  MoveL 7361 to (552.16, 514.95, 128) mm, rotated rx 180 ry 0 rz 160 deg; joints [7.263, 67.715, -20.224, -145.045, 53.083, 157.223]
  Set speed (16.3 mm/s)
  Call Extruder(797.85482)
  MoveL 7362 to (551.52, 517.03, 128) mm, rotated rx -180 ry 0 rz 160 deg; joints [7.506, 67.637, -20.071, -144.797, 53.24, 157.109]
  Call Extruder(805.35406)
  MoveL 7363 to (550.8, 519.07, 128) mm, rotated rx 180 ry 0 rz 160 deg; joints [7.746, 67.545, -19.889, -144.56, 53.407, 157.01]
  Set speed (16.3 mm/s)
  Call Extruder(809.35775)
  MoveL 7364 to (550.38, 520.14, 128) mm, rotated rx 180 ry 0 rz 160 deg; joints [7.874, 67.489, -19.778, -144.438, 53.501, 156.962]
  Set speed (16.2 mm/s)
  Call Extruder(812.97522)
  MoveL 7365 to (549.99, 521.11, 128) mm, rotated rx 180 ry 0 rz 160 deg; joints [7.988, 67.436, -19.673, -144.329, 53.588, 156.922]
  Set speed (16.2 mm/s)
  Call Extruder(817.04856)
  MoveL 7366 to (549.52, 522.18, 128) mm, rotated rx 180 ry 0 rz 160 deg; joints [8.117, 67.37, -19.543, -144.21, 53.691, 156.882]
  Set speed (16.3 mm/s)
  Call Extruder(820.74398)
  MoveL 7367 to (549.08, 523.15, 128) mm, rotated rx 180 ry 0 rz 160 deg; joints [8.233, 67.308, -19.421, -144.103, 53.786, 156.847]
  Set speed (16.3 mm/s)
  Call Extruder(824.78698)
  MoveL 7368 to (548.57, 524.2, 128) mm, rotated rx -180 ry 0 rz 160 deg; joints [8.359, 67.236, -19.278, -143.989, 53.893, 156.814]
  Set speed (16.3 mm/s)
  Call Extruder(830.04096)
  MoveL 7369 to (547.87, 525.55, 128) mm, rotated rx 180 ry 0 rz 160 deg; joints [8.523, 67.135, -19.079, -143.846, 54.037, 156.776]
  Set speed (16.3 mm/s)
  Call Extruder(836.18149)
  MoveL 7370 to (547.01, 527.1, 128) mm, rotated rx 180 ry 0 rz 160 deg; joints [8.712, 67.009, -18.828, -143.684, 54.212, 156.741]
  Set speed (16.3 mm/s)
  Call Extruder(840.06133)
  MoveL 7371 to (546.44, 528.06, 128) mm, rotated rx 180 ry 0 rz 160 deg; joints [8.831, 66.924, -18.66, -143.585, 54.325, 156.723]
  Set speed (16.3 mm/s)
  Call Extruder(844.64327)
  MoveL 7372 to (545.75, 529.18, 128) mm, rotated rx 180 ry 0 rz 160 deg; joints [8.97, 66.819, -18.453, -143.472, 54.463, 156.707]
  Set speed (16.3 mm/s)
  Call Extruder(847.13279)
  MoveL 7373 to (545.36, 529.78, 128) mm, rotated rx -180 ry 0 rz 160 deg; joints [9.045, 66.761, -18.336, -143.412, 54.539, 156.7]
  Set speed (16.3 mm/s)
  Call Extruder(851.62819)
  MoveL 7374 to (544.63, 530.86, 128) mm, rotated rx 180 ry 0 rz 160 deg; joints [9.179, 66.65, -18.117, -143.306, 54.679, 156.692]
  Set speed (16.3 mm/s)
  Call Extruder(855.44742)
  MoveL 7375 to (544, 531.76, 128) mm, rotated rx -180 ry 0 rz 160 deg; joints [9.293, 66.553, -17.924, -143.219, 54.801, 156.688]
  Set speed (16.3 mm/s)
  Call Extruder(859.46697)
  MoveL 7376 to (543.31, 532.69, 128) mm, rotated rx 180 ry 0 rz 160 deg; joints [9.411, 66.446, -17.713, -143.13, 54.931, 156.688]
  Set speed (16.3 mm/s)
  Call Extruder(863.24458)
  MoveL 7377 to (542.65, 533.55, 128) mm, rotated rx 180 ry 0 rz 160 deg; joints [9.522, 66.344, -17.51, -143.049, 55.055, 156.691]
  Set speed (16.3 mm/s)
  Call Extruder(867.09312)
  MoveL 7378 to (541.95, 534.42, 128) mm, rotated rx -180 ry 0 rz 160 deg; joints [9.633, 66.235, -17.295, -142.969, 55.185, 156.698]
  Set speed (16.3 mm/s)
  Call Extruder(870.82681)
  MoveL 7379 to (541.26, 535.24, 128) mm, rotated rx -180 ry 0 rz 160 deg; joints [9.74, 66.128, -17.082, -142.894, 55.311, 156.707]
  Set speed (16.3 mm/s)
  Call Extruder(874.69315)
  MoveL 7380 to (540.53, 536.08, 128) mm, rotated rx 180 ry 0 rz 160 deg; joints [9.85, 66.013, -16.854, -142.818, 55.445, 156.721]
  Set speed (16.3 mm/s)
  Call Extruder(878.56523)
  MoveL 7381 to (539.77, 536.91, 128) mm, rotated rx -180 ry 0 rz 160 deg; joints [9.958, 65.895, -16.619, -142.746, 55.58, 156.737]
  Call Extruder(882.39538)
  MoveL 7382 to (539.02, 537.71, 128) mm, rotated rx -180 ry 0 rz 160 deg; joints [10.065, 65.775, -16.382, -142.676, 55.716, 156.757]
  Call Extruder(886.34677)
  MoveL 7383 to (538.22, 538.52, 128) mm, rotated rx -180 ry 0 rz 160 deg; joints [10.173, 65.649, -16.131, -142.607, 55.858, 156.781]
  Set speed (16.3 mm/s)
  Call Extruder(890.12986)
  MoveL 7384 to (537.43, 539.28, 128) mm, rotated rx 180 ry 0 rz 160 deg; joints [10.276, 65.525, -15.885, -142.543, 55.996, 156.807]
  Call Extruder(893.94691)
  MoveL 7385 to (536.63, 540.03, 128) mm, rotated rx -180 ry 0 rz 160 deg; joints [10.378, 65.398, -15.631, -142.482, 56.136, 156.836]
  Call Extruder(897.84566)
  MoveL 7386 to (535.79, 540.78, 128) mm, rotated rx -180 ry 0 rz 160 deg; joints [10.481, 65.265, -15.367, -142.421, 56.28, 156.869]
  Set speed (16.3 mm/s)
  Call Extruder(901.21524)
  MoveL 7387 to (535.06, 541.42, 128) mm, rotated rx 180 ry 0 rz 160 deg; joints [10.57, 65.148, -15.135, -142.37, 56.407, 156.899]
  Set speed (16.3 mm/s)
  Call Extruder(905.50699)
  MoveL 7388 to (534.11, 542.2, 128) mm, rotated rx -180 ry 0 rz 160 deg; joints [10.68, 64.996, -14.833, -142.309, 56.569, 156.942]
  Set speed (16.3 mm/s)
  Call Extruder(908.78682)
  MoveL 7389 to (533.36, 542.79, 128) mm, rotated rx 180 ry 0 rz 160 deg; joints [10.763, 64.878, -14.597, -142.265, 56.694, 156.978]
  Set speed (16.3 mm/s)
  Call Extruder(913.16892)
  MoveL 7390 to (532.36, 543.56, 128) mm, rotated rx 180 ry 0 rz 160 deg; joints [10.873, 64.718, -14.278, -142.208, 56.862, 157.027]
  Call Extruder(917.07721)
  MoveL 7391 to (531.45, 544.22, 128) mm, rotated rx 180 ry 0 rz 160 deg; joints [10.969, 64.572, -13.988, -142.16, 57.014, 157.075]
  Set speed (16.3 mm/s)
  Call Extruder(920.88896)
  MoveL 7392 to (530.55, 544.85, 128) mm, rotated rx -180 ry 0 rz 160 deg; joints [11.061, 64.428, -13.701, -142.115, 57.163, 157.125]
  Set speed (16.3 mm/s)
  Call Extruder(924.82440)
  MoveL 7393 to (529.6, 545.48, 128) mm, rotated rx 180 ry 0 rz 160 deg; joints [11.155, 64.277, -13.4, -142.072, 57.318, 157.179]
  Set speed (16.3 mm/s)
  Call Extruder(928.58871)
  MoveL 7394 to (528.69, 546.06, 128) mm, rotated rx -180 ry 0 rz 160 deg; joints [11.243, 64.13, -13.108, -142.033, 57.467, 157.233]
  Set speed (16.3 mm/s)
  Call Extruder(932.50029)
  MoveL 7395 to (527.73, 546.64, 128) mm, rotated rx -180 ry 0 rz 160 deg; joints [11.333, 63.976, -12.8, -141.994, 57.622, 157.293]
  Set speed (16.3 mm/s)
  Call Extruder(936.32920)
  MoveL 7396 to (526.77, 547.2, 128) mm, rotated rx 180 ry 0 rz 160 deg; joints [11.419, 63.823, -12.495, -141.96, 57.775, 157.353]
  Set speed (16.3 mm/s)
  Call Extruder(939.88963)
  MoveL 7397 to (525.88, 547.7, 128) mm, rotated rx -180 ry 0 rz 160 deg; joints [11.498, 63.679, -12.208, -141.929, 57.918, 157.412]
  Set speed (16.3 mm/s)
  Call Extruder(946.13638)
  MoveL 7398 to (524.28, 548.53, 128) mm, rotated rx 180 ry 0 rz 160 deg; joints [11.632, 63.424, -11.698, -141.881, 58.17, 157.52]
  Call Extruder(951.88293)
  MoveL 7399 to (522.79, 549.25, 128) mm, rotated rx 180 ry 0 rz 160 deg; joints [11.751, 63.185, -11.22, -141.843, 58.404, 157.625]
  Set speed (16.3 mm/s)
  Call Extruder(959.39188)
  MoveL 7400 to (520.81, 550.12, 128) mm, rotated rx 180 ry 0 rz 160 deg; joints [11.901, 62.867, -10.585, -141.8, 58.71, 157.77]
  Call Extruder(967.32682)
  MoveL 7401 to (518.68, 550.95, 128) mm, rotated rx 180 ry 0 rz 160 deg; joints [12.051, 62.526, -9.902, -141.766, 59.035, 157.933]
  Set speed (16.3 mm/s)
  Call Extruder(974.78424)
  MoveL 7402 to (516.64, 551.64, 128) mm, rotated rx 180 ry 0 rz 160 deg; joints [12.184, 62.2, -9.25, -141.743, 59.341, 158.095]
  Set speed (16.2 mm/s)
  Call Extruder(978.78034)
  MoveL 7403 to (515.54, 551.98, 128) mm, rotated rx -180 ry 0 rz 160 deg; joints [12.252, 62.024, -8.897, -141.734, 59.505, 158.185]
  Set speed (16.3 mm/s)
  Call Extruder(982.65084)
  MoveL 7404 to (514.48, 552.3, 128) mm, rotated rx 180 ry 0 rz 160 deg; joints [12.316, 61.854, -8.554, -141.727, 59.664, 158.273]
  Call Extruder(985.91733)
  MoveL 7405 to (513.56, 552.54, 128) mm, rotated rx -180 ry 0 rz 160 deg; joints [12.368, 61.708, -8.262, -141.725, 59.798, 158.351]
  Set speed (16.2 mm/s)
  Call Extruder(990.16839)
  MoveL 7406 to (512.38, 552.83, 128) mm, rotated rx -180 ry 0 rz 160 deg; joints [12.434, 61.518, -7.881, -141.723, 59.973, 158.452]
  Set speed (16.3 mm/s)
  Call Extruder(998.02753)
  MoveL 7407 to (510.16, 553.3, 128) mm, rotated rx 180 ry 0 rz 160 deg; joints [12.548, 61.165, -7.171, -141.727, 60.295, 158.646]
  Set speed (16.3 mm/s)
  Call Extruder(1005.81110)
  MoveL 7408 to (507.95, 553.68, 128) mm, rotated rx 180 ry 0 rz 160 deg; joints [12.652, 60.812, -6.461, -141.742, 60.612, 158.845]
  Call Extruder(1013.42033)
  MoveL 7409 to (505.77, 553.95, 128) mm, rotated rx -180 ry 0 rz 160 deg; joints [12.743, 60.464, -5.762, -141.766, 60.921, 159.047]
  Set speed (16.3 mm/s)
  Call Extruder(1021.17666)
  MoveL 7410 to (503.55, 554.15, 128) mm, rotated rx 180 ry 0 rz 160 deg; joints [12.827, 60.109, -5.047, -141.799, 61.234, 159.258]
  Set speed (16.3 mm/s)
  Call Extruder(1028.91579)
  MoveL 7411 to (501.32, 554.25, 128) mm, rotated rx 180 ry 0 rz 160 deg; joints [12.9, 59.754, -4.33, -141.843, 61.544, 159.475]
  Set speed (16.3 mm/s)
  Call Extruder(1036.52400)
  MoveL 7412 to (499.12, 554.25, 128) mm, rotated rx 180 ry 0 rz 160 deg; joints [12.962, 59.405, -3.625, -141.895, 61.846, 159.694]
  Set speed (10.0 mm/s)
  MoveL 7413 to (499.12, 554.25, 132) mm, rotated rx 180 ry 0 rz 160 deg; joints [12.962, 58.806, -3.422, -141.763, 61.534, 159.416]
  Set speed (120.0 mm/s)
  MoveL 7414 to (499.15, 552.4, 132) mm, rotated rx 180 ry 0 rz 160 deg; joints [12.736, 58.744, -3.297, -142.025, 61.505, 159.575]
  Set speed (16.4 mm/s)
  Call Extruder(1043.97760)
  MoveL 7415 to (496.99, 552.32, 132) mm, rotated rx 180 ry 0 rz 160 deg; joints [12.786, 58.398, -2.602, -142.088, 61.797, 159.793]
  Set speed (16.4 mm/s)
  Call Extruder(1051.39615)
  MoveL 7416 to (494.85, 552.15, 132) mm, rotated rx 180 ry 0 rz 160 deg; joints [12.825, 58.055, -1.913, -142.16, 62.084, 160.015]
  Call Extruder(1058.70817)
  MoveL 7417 to (492.74, 551.9, 132) mm, rotated rx 180 ry 0 rz 160 deg; joints [12.853, 57.719, -1.235, -142.24, 62.364, 160.237]
  Set speed (16.4 mm/s)
  Call Extruder(1066.06150)
  MoveL 7418 to (490.64, 551.56, 132) mm, rotated rx -180 ry 0 rz 160 deg; joints [12.871, 57.381, -0.555, -142.331, 62.64, 160.465]
  Set speed (16.4 mm/s)
  Call Extruder(1073.73360)
  MoveL 7419 to (488.45, 551.12, 132) mm, rotated rx 180 ry 0 rz 160 deg; joints [12.878, 57.032, 0.149, -142.435, 62.924, 160.705]
  Set speed (16.4 mm/s)
  Call Extruder(1077.22198)
  MoveL 7420 to (487.47, 550.88, 132) mm, rotated rx -180 ry 0 rz 160 deg; joints [12.876, 56.874, 0.467, -142.486, 63.051, 160.816]
  Call Extruder(1080.67093)
  MoveL 7421 to (486.5, 550.64, 132) mm, rotated rx -180 ry 0 rz 160 deg; joints [12.873, 56.719, 0.781, -142.538, 63.175, 160.925]
  Set speed (16.4 mm/s)
  Call Extruder(1084.57071)
  MoveL 7422 to (485.41, 550.33, 132) mm, rotated rx -180 ry 0 rz 160 deg; joints [12.866, 56.545, 1.134, -142.6, 63.314, 161.05]
  Call Extruder(1088.21611)
  MoveL 7423 to (484.4, 550.03, 132) mm, rotated rx 180 ry 0 rz 160 deg; joints [12.857, 56.382, 1.462, -142.66, 63.443, 161.167]
  Set speed (16.4 mm/s)
  Call Extruder(1095.48451)
  MoveL 7424 to (482.4, 549.36, 132) mm, rotated rx 180 ry 0 rz 160 deg; joints [12.831, 56.061, 2.112, -142.787, 63.697, 161.402]
  Set speed (16.4 mm/s)
  Call Extruder(1099.40980)
  MoveL 7425 to (481.33, 548.96, 132) mm, rotated rx 180 ry 0 rz 160 deg; joints [12.811, 55.889, 2.46, -142.86, 63.83, 161.529]
  Set speed (16.4 mm/s)
  Call Extruder(1103.58260)
  MoveL 7426 to (480.21, 548.52, 132) mm, rotated rx 180 ry 0 rz 160 deg; joints [12.788, 55.708, 2.827, -142.94, 63.971, 161.665]
  Set speed (16.3 mm/s)
  Call Extruder(1108.58819)
  MoveL 7427 to (478.87, 547.96, 132) mm, rotated rx -180 ry 0 rz 160 deg; joints [12.755, 55.493, 3.263, -143.04, 64.137, 161.828]
  Set speed (16.4 mm/s)
  Call Extruder(1114.05266)
  MoveL 7428 to (477.43, 547.3, 132) mm, rotated rx 180 ry 0 rz 160 deg; joints [12.712, 55.26, 3.734, -143.154, 64.315, 162.007]
  Set speed (16.4 mm/s)
  Call Extruder(1117.85423)
  MoveL 7429 to (476.44, 546.81, 132) mm, rotated rx -180 ry 0 rz 160 deg; joints [12.678, 55.1, 4.06, -143.237, 64.437, 162.132]
  Set speed (16.4 mm/s)
  Call Extruder(1121.57728)
  MoveL 7430 to (475.48, 546.32, 132) mm, rotated rx 180 ry 0 rz 160 deg; joints [12.642, 54.945, 4.375, -143.321, 64.554, 162.255]
  Set speed (16.4 mm/s)
  Call Extruder(1124.36398)
  MoveL 7431 to (474.77, 545.93, 132) mm, rotated rx -180 ry 0 rz 160 deg; joints [12.613, 54.829, 4.61, -143.385, 64.641, 162.346]
  Set speed (16.4 mm/s)
  Call Extruder(1128.80316)
  MoveL 7432 to (473.65, 545.3, 132) mm, rotated rx 180 ry 0 rz 160 deg; joints [12.564, 54.647, 4.98, -143.49, 64.777, 162.493]
  Call Extruder(1132.57278)
  MoveL 7433 to (472.71, 544.74, 132) mm, rotated rx -180 ry 0 rz 160 deg; joints [12.518, 54.494, 5.291, -143.582, 64.891, 162.617]
  Set speed (16.4 mm/s)
  Call Extruder(1136.28054)
  MoveL 7434 to (471.79, 544.17, 132) mm, rotated rx -180 ry 0 rz 160 deg; joints [12.471, 54.346, 5.593, -143.675, 65.001, 162.739]
  Call Extruder(1139.90076)
  MoveL 7435 to (470.92, 543.59, 132) mm, rotated rx 180 ry 0 rz 160 deg; joints [12.421, 54.202, 5.885, -143.768, 65.106, 162.858]
  Set speed (16.4 mm/s)
  Call Extruder(1143.59875)
  MoveL 7436 to (470.03, 542.99, 132) mm, rotated rx 180 ry 0 rz 160 deg; joints [12.368, 54.057, 6.181, -143.865, 65.211, 162.979]
  Set speed (16.4 mm/s)
  Call Extruder(1147.38632)
  MoveL 7437 to (469.13, 542.35, 132) mm, rotated rx -180 ry 0 rz 160 deg; joints [12.31, 53.911, 6.479, -143.968, 65.317, 163.103]
  Set speed (16.4 mm/s)
  Call Extruder(1150.96414)
  MoveL 7438 to (468.3, 541.73, 132) mm, rotated rx 180 ry 0 rz 160 deg; joints [12.253, 53.774, 6.758, -144.066, 65.416, 163.22]
  Set speed (16.4 mm/s)
  Call Extruder(1154.80847)
  MoveL 7439 to (467.42, 541.05, 132) mm, rotated rx 180 ry 0 rz 160 deg; joints [12.188, 53.629, 7.054, -144.174, 65.519, 163.346]
  Call Extruder(1158.41047)
  MoveL 7440 to (466.61, 540.39, 132) mm, rotated rx 180 ry 0 rz 160 deg; joints [12.124, 53.495, 7.327, -144.279, 65.614, 163.463]
  Call Extruder(1162.10973)
  MoveL 7441 to (465.79, 539.69, 132) mm, rotated rx -180 ry 0 rz 160 deg; joints [12.056, 53.36, 7.604, -144.387, 65.71, 163.583]
  Set speed (16.4 mm/s)
  Call Extruder(1165.90163)
  MoveL 7442 to (464.96, 538.97, 132) mm, rotated rx 180 ry 0 rz 160 deg; joints [11.984, 53.222, 7.884, -144.501, 65.806, 163.705]
  Set speed (16.4 mm/s)
  Call Extruder(1169.28030)
  MoveL 7443 to (464.24, 538.31, 132) mm, rotated rx 180 ry 0 rz 160 deg; joints [11.916, 53.102, 8.13, -144.605, 65.889, 163.814]
  Set speed (16.4 mm/s)
  Call Extruder(1172.26831)
  MoveL 7444 to (463.61, 537.71, 132) mm, rotated rx -180 ry 0 rz 160 deg; joints [11.854, 52.998, 8.344, -144.698, 65.961, 163.91]
  Set speed (16.4 mm/s)
  Call Extruder(1176.91926)
  MoveL 7445 to (462.65, 536.76, 132) mm, rotated rx -180 ry 0 rz 160 deg; joints [11.754, 52.838, 8.671, -144.846, 66.07, 164.059]
  Set speed (16.4 mm/s)
  Call Extruder(1180.58115)
  MoveL 7446 to (461.91, 535.99, 132) mm, rotated rx 180 ry 0 rz 160 deg; joints [11.673, 52.714, 8.925, -144.965, 66.154, 164.175]
  Set speed (16.4 mm/s)
  Call Extruder(1184.31373)
  MoveL 7447 to (461.17, 535.2, 132) mm, rotated rx 180 ry 0 rz 160 deg; joints [11.587, 52.59, 9.178, -145.088, 66.237, 164.293]
  Set speed (16.4 mm/s)
  Call Extruder(1187.19569)
  MoveL 7448 to (460.62, 534.57, 132) mm, rotated rx -180 ry 0 rz 160 deg; joints [11.518, 52.496, 9.371, -145.185, 66.299, 164.383]
  Set speed (16.4 mm/s)
  Call Extruder(1191.17044)
  MoveL 7449 to (459.87, 533.7, 132) mm, rotated rx 180 ry 0 rz 160 deg; joints [11.421, 52.369, 9.632, -145.321, 66.383, 164.507]
  Set speed (16.4 mm/s)
  Call Extruder(1195.44747)
  MoveL 7450 to (459.08, 532.74, 132) mm, rotated rx -180 ry 0 rz 160 deg; joints [11.313, 52.235, 9.906, -145.469, 66.47, 164.64]
  Set speed (16.4 mm/s)
  Call Extruder(1199.06168)
  MoveL 7451 to (458.43, 531.91, 132) mm, rotated rx 180 ry 0 rz 160 deg; joints [11.219, 52.124, 10.133, -145.597, 66.541, 164.751]
  Call Extruder(1202.74625)
  MoveL 7452 to (457.79, 531.06, 132) mm, rotated rx 180 ry 0 rz 160 deg; joints [11.121, 52.014, 10.359, -145.729, 66.611, 164.864]
  Set speed (16.4 mm/s)
  Call Extruder(1206.43074)
  MoveL 7453 to (457.17, 530.19, 132) mm, rotated rx 180 ry 0 rz 160 deg; joints [11.02, 51.906, 10.581, -145.863, 66.679, 164.975]
  Set speed (16.4 mm/s)
  Call Extruder(1210.21210)
  MoveL 7454 to (456.55, 529.29, 132) mm, rotated rx -180 ry 0 rz 160 deg; joints [10.913, 51.798, 10.803, -146.002, 66.746, 165.089]
  Set speed (16.4 mm/s)
  Call Extruder(1213.92244)
  MoveL 7455 to (455.95, 528.39, 132) mm, rotated rx 180 ry 0 rz 160 deg; joints [10.806, 51.695, 11.015, -146.141, 66.809, 165.2]
  Set speed (16.4 mm/s)
  Call Extruder(1217.52902)
  MoveL 7456 to (455.39, 527.51, 132) mm, rotated rx -180 ry 0 rz 160 deg; joints [10.7, 51.597, 11.217, -146.277, 66.868, 165.306]
  Set speed (16.4 mm/s)
  Call Extruder(1221.90125)
  MoveL 7457 to (454.74, 526.42, 132) mm, rotated rx -180 ry 0 rz 160 deg; joints [10.568, 51.482, 11.454, -146.445, 66.936, 165.434]
  Call Extruder(1228.58017)
  MoveL 7458 to (453.79, 524.73, 132) mm, rotated rx -180 ry 0 rz 160 deg; joints [10.359, 51.313, 11.802, -146.706, 67.033, 165.627]
  Set speed (16.4 mm/s)
  Call Extruder(1232.29007)
  MoveL 7459 to (453.3, 523.77, 132) mm, rotated rx -180 ry 0 rz 160 deg; joints [10.241, 51.223, 11.987, -146.853, 67.083, 165.732]
  Call Extruder(1236.08269)
  MoveL 7460 to (452.81, 522.79, 132) mm, rotated rx -180 ry 0 rz 160 deg; joints [10.117, 51.134, 12.17, -147.005, 67.132, 165.839]
  Set speed (16.4 mm/s)
  Call Extruder(1243.24840)
  MoveL 7461 to (451.94, 520.9, 132) mm, rotated rx 180 ry 0 rz 160 deg; joints [9.876, 50.974, 12.5, -147.297, 67.216, 166.037]
  Set speed (16.4 mm/s)
  Call Extruder(1247.17185)
  MoveL 7462 to (451.5, 519.85, 132) mm, rotated rx -180 ry 0 rz 160 deg; joints [9.741, 50.891, 12.67, -147.459, 67.258, 166.143]
  Set speed (16.4 mm/s)
  Call Extruder(1250.87077)
  MoveL 7463 to (451.1, 518.85, 132) mm, rotated rx 180 ry 0 rz 160 deg; joints [9.612, 50.815, 12.827, -147.613, 67.295, 166.243]
  Set speed (16.4 mm/s)
  Call Extruder(1254.56538)
  MoveL 7464 to (450.73, 517.85, 132) mm, rotated rx 180 ry 0 rz 160 deg; joints [9.481, 50.744, 12.974, -147.768, 67.328, 166.34]
  Set speed (16.4 mm/s)
  Call Extruder(1258.09802)
  MoveL 7465 to (450.39, 516.88, 132) mm, rotated rx 180 ry 0 rz 160 deg; joints [9.354, 50.677, 13.112, -147.917, 67.358, 166.432]
  Set speed (16.4 mm/s)
  Call Extruder(1261.95788)
  MoveL 7466 to (450.05, 515.82, 132) mm, rotated rx 180 ry 0 rz 160 deg; joints [9.214, 50.608, 13.254, -148.082, 67.387, 166.531]
  Set speed (16.4 mm/s)
  Call Extruder(1265.49475)
  MoveL 7467 to (449.74, 514.84, 132) mm, rotated rx -180 ry 0 rz 160 deg; joints [9.084, 50.547, 13.38, -148.233, 67.413, 166.621]
  Set speed (16.4 mm/s)
  Call Extruder(1272.94487)
  MoveL 7468 to (449.17, 512.75, 132) mm, rotated rx -180 ry 0 rz 160 deg; joints [8.804, 50.429, 13.625, -148.555, 67.456, 166.806]
  Set speed (16.4 mm/s)
  Call Extruder(1280.31638)
  MoveL 7469 to (448.69, 510.67, 132) mm, rotated rx -180 ry 0 rz 160 deg; joints [8.521, 50.324, 13.842, -148.878, 67.488, 166.984]
  Set speed (16.4 mm/s)
  Call Extruder(1287.84373)
  MoveL 7470 to (448.29, 508.52, 132) mm, rotated rx 180 ry 0 rz 160 deg; joints [8.226, 50.229, 14.038, -149.21, 67.508, 167.159]
  Call Extruder(1295.22150)
  MoveL 7471 to (447.99, 506.4, 132) mm, rotated rx 180 ry 0 rz 160 deg; joints [7.933, 50.15, 14.202, -149.538, 67.517, 167.324]
  Set speed (16.4 mm/s)
  Call Extruder(1302.60966)
  MoveL 7472 to (447.77, 504.27, 132) mm, rotated rx -180 ry 0 rz 160 deg; joints [7.635, 50.082, 14.341, -149.867, 67.514, 167.484]
  Set speed (16.4 mm/s)
  Call Extruder(1309.81071)
  MoveL 7473 to (447.64, 502.18, 132) mm, rotated rx 180 ry 0 rz 160 deg; joints [7.342, 50.03, 14.45, -150.189, 67.499, 167.633]
  Set speed (16.4 mm/s)
  Call Extruder(1317.28696)
  MoveL 7474 to (447.59, 500.01, 132) mm, rotated rx -180 ry 0 rz 160 deg; joints [7.034, 49.988, 14.537, -150.524, 67.473, 167.781]
  Set speed (16.4 mm/s)
  Call Extruder(1324.02628)
  MoveL 7475 to (447.63, 498.06, 132) mm, rotated rx 180 ry 0 rz 160 deg; joints [6.755, 49.962, 14.591, -150.824, 67.439, 167.909]
  Set speed (16.4 mm/s)
  Call Extruder(1330.58179)
  MoveL 7476 to (447.74, 496.16, 132) mm, rotated rx 180 ry 0 rz 160 deg; joints [6.483, 49.947, 14.622, -151.116, 67.396, 168.028]
  Set speed (16.4 mm/s)
  Call Extruder(1337.23196)
  MoveL 7477 to (447.91, 494.24, 132) mm, rotated rx -180 ry 0 rz 160 deg; joints [6.206, 49.941, 14.634, -151.41, 67.344, 168.144]
  Call Extruder(1343.87995)
  MoveL 7478 to (448.16, 492.32, 132) mm, rotated rx 180 ry 0 rz 160 deg; joints [5.93, 49.947, 14.621, -151.703, 67.282, 168.254]
  Set speed (16.4 mm/s)
  Call Extruder(1350.61226)
  MoveL 7479 to (448.48, 490.4, 132) mm, rotated rx 180 ry 0 rz 160 deg; joints [5.65, 49.964, 14.586, -151.996, 67.209, 168.36]
  Set speed (16.4 mm/s)
  Call Extruder(1357.16591)
  MoveL 7480 to (448.86, 488.53, 132) mm, rotated rx -180 ry 0 rz 160 deg; joints [5.379, 49.991, 14.531, -152.278, 67.13, 168.457]
  Set speed (16.4 mm/s)
  Call Extruder(1363.73554)
  MoveL 7481 to (449.31, 486.68, 132) mm, rotated rx 180 ry 0 rz 160 deg; joints [5.109, 50.028, 14.455, -152.558, 67.041, 168.549]
  Set speed (16.4 mm/s)
  Call Extruder(1370.46103)
  MoveL 7482 to (449.85, 484.8, 132) mm, rotated rx -180 ry 0 rz 160 deg; joints [4.835, 50.076, 14.354, -152.84, 66.94, 168.637]
  Call Extruder(1377.10545)
  MoveL 7483 to (450.44, 482.97, 132) mm, rotated rx 180 ry 0 rz 160 deg; joints [4.567, 50.135, 14.233, -153.114, 66.832, 168.719]
  Set speed (16.4 mm/s)
  Call Extruder(1383.92639)
  MoveL 7484 to (451.12, 481.11, 132) mm, rotated rx -180 ry 0 rz 160 deg; joints [4.294, 50.206, 14.086, -153.39, 66.711, 168.796]
  Set speed (16.4 mm/s)
  Call Extruder(1389.57705)
  MoveL 7485 to (451.73, 479.59, 132) mm, rotated rx 180 ry 0 rz 160 deg; joints [4.072, 50.272, 13.949, -153.614, 66.604, 168.856]
  Set speed (16.4 mm/s)
  Call Extruder(1396.98627)
  MoveL 7486 to (452.61, 477.63, 132) mm, rotated rx 180 ry 0 rz 160 deg; joints [3.785, 50.371, 13.744, -153.901, 66.454, 168.927]
  Set speed (16.4 mm/s)
  Call Extruder(1403.53462)
  MoveL 7487 to (453.45, 475.93, 132) mm, rotated rx 180 ry 0 rz 160 deg; joints [3.535, 50.469, 13.542, -154.148, 66.313, 168.984]
  Set speed (16.4 mm/s)
  Call Extruder(1410.46010)
  MoveL 7488 to (454.41, 474.16, 132) mm, rotated rx -180 ry 0 rz 160 deg; joints [3.277, 50.583, 13.307, -154.402, 66.154, 169.039]
  Set speed (16.4 mm/s)
  Call Extruder(1417.00264)
  MoveL 7489 to (455.38, 472.52, 132) mm, rotated rx -180 ry 0 rz 160 deg; joints [3.038, 50.7, 13.065, -154.634, 65.996, 169.084]
  Set speed (16.4 mm/s)
  Call Extruder(1423.55518)
  MoveL 7490 to (456.4, 470.92, 132) mm, rotated rx -180 ry 0 rz 160 deg; joints [2.805, 50.827, 12.803, -154.859, 65.83, 169.123]
  Set speed (16.4 mm/s)
  Call Extruder(1430.30707)
  MoveL 7491 to (457.52, 469.31, 132) mm, rotated rx 180 ry 0 rz 160 deg; joints [2.571, 50.967, 12.513, -155.083, 65.65, 169.157]
  Set speed (16.4 mm/s)
  Call Extruder(1437.04503)
  MoveL 7492 to (458.69, 467.75, 132) mm, rotated rx 180 ry 0 rz 160 deg; joints [2.345, 51.117, 12.204, -155.297, 65.464, 169.185]
  Set speed (16.4 mm/s)
  Call Extruder(1443.60356)
  MoveL 7493 to (459.89, 466.27, 132) mm, rotated rx -180 ry 0 rz 160 deg; joints [2.131, 51.272, 11.885, -155.496, 65.274, 169.206]
  Set speed (16.4 mm/s)
  Call Extruder(1450.24651)
  MoveL 7494 to (461.16, 464.82, 132) mm, rotated rx -180 ry 0 rz 160 deg; joints [1.922, 51.438, 11.544, -155.689, 65.075, 169.221]
  Call Extruder(1456.99716)
  MoveL 7495 to (462.5, 463.39, 132) mm, rotated rx 180 ry 0 rz 160 deg; joints [1.718, 51.615, 11.179, -155.875, 64.866, 169.23]
  Set speed (16.4 mm/s)
  Call Extruder(1463.55215)
  MoveL 7496 to (463.86, 462.05, 132) mm, rotated rx -180 ry 0 rz 160 deg; joints [1.527, 51.796, 10.807, -156.045, 64.656, 169.232]
  Call Extruder(1470.23484)
  MoveL 7497 to (465.28, 460.74, 132) mm, rotated rx 180 ry 0 rz 160 deg; joints [1.34, 51.989, 10.412, -156.209, 64.436, 169.229]
  Call Extruder(1476.72745)
  MoveL 7498 to (466.72, 459.52, 132) mm, rotated rx 180 ry 0 rz 160 deg; joints [1.167, 52.184, 10.011, -156.358, 64.215, 169.219]
  Set speed (16.4 mm/s)
  Call Extruder(1483.94711)
  MoveL 7499 to (468.36, 458.22, 132) mm, rotated rx 180 ry 0 rz 160 deg; joints [0.985, 52.409, 9.548, -156.511, 63.964, 169.2]
  Set speed (16.4 mm/s)
  Call Extruder(1490.19198)
  MoveL 7500 to (469.83, 457.15, 132) mm, rotated rx 180 ry 0 rz 160 deg; joints [0.835, 52.612, 9.133, -156.633, 63.741, 169.178]
  Set speed (16.4 mm/s)
  Call Extruder(1496.79061)
  MoveL 7501 to (471.41, 456.08, 132) mm, rotated rx -180 ry 0 rz 160 deg; joints [0.686, 52.833, 8.68, -156.752, 63.5, 169.149]
  Set speed (16.4 mm/s)
  Call Extruder(1503.52368)
  MoveL 7502 to (473.07, 455.05, 132) mm, rotated rx 180 ry 0 rz 160 deg; joints [0.543, 53.066, 8.204, -156.861, 63.249, 169.112]
  Set speed (16.4 mm/s)
  Call Extruder(1510.17787)
  MoveL 7503 to (474.74, 454.09, 132) mm, rotated rx 180 ry 0 rz 160 deg; joints [0.411, 53.303, 7.719, -156.957, 62.996, 169.069]
  Set speed (16.4 mm/s)
  Call Extruder(1516.77838)
  MoveL 7504 to (476.44, 453.19, 132) mm, rotated rx 180 ry 0 rz 160 deg; joints [0.289, 53.545, 7.226, -157.041, 62.741, 169.019]
  Call Extruder(1523.42900)
  MoveL 7505 to (478.18, 452.36, 132) mm, rotated rx 180 ry 0 rz 160 deg; joints [0.176, 53.795, 6.716, -157.113, 62.48, 168.963]
  Set speed (16.4 mm/s)
  Call Extruder(1530.12968)
  MoveL 7506 to (479.96, 451.58, 132) mm, rotated rx 180 ry 0 rz 160 deg; joints [0.071, 54.052, 6.19, -157.175, 62.213, 168.899]
  Set speed (16.4 mm/s)
  Call Extruder(1536.60605)
  MoveL 7507 to (481.71, 450.89, 132) mm, rotated rx 180 ry 0 rz 160 deg; joints [-0.02, 54.307, 5.671, -157.222, 61.952, 168.831]
  Set speed (16.4 mm/s)
  Call Extruder(1543.43975)
  MoveL 7508 to (483.58, 450.24, 132) mm, rotated rx 180 ry 0 rz 160 deg; joints [-0.107, 54.582, 5.113, -157.26, 61.673, 168.752]
  Set speed (16.4 mm/s)
  Call Extruder(1550.03230)
  MoveL 7509 to (485.4, 449.67, 132) mm, rotated rx 180 ry 0 rz 160 deg; joints [-0.181, 54.851, 4.565, -157.284, 61.402, 168.669]
  Set speed (16.4 mm/s)
  Call Extruder(1556.62361)
  MoveL 7510 to (487.25, 449.17, 132) mm, rotated rx 180 ry 0 rz 160 deg; joints [-0.246, 55.126, 4.007, -157.297, 61.128, 168.579]
  Set speed (16.4 mm/s)
  Call Extruder(1563.37623)
  MoveL 7511 to (489.16, 448.73, 132) mm, rotated rx -180 ry 0 rz 160 deg; joints [-0.303, 55.412, 3.427, -157.297, 60.845, 168.48]
  Set speed (16.4 mm/s)
  Call Extruder(1569.85466)
  MoveL 7512 to (491.01, 448.37, 132) mm, rotated rx 180 ry 0 rz 160 deg; joints [-0.347, 55.69, 2.863, -157.286, 60.573, 168.378]
  Call Extruder(0.00000)
  Set speed (16.4 mm/s)
  Call Extruder(6.52179)
  MoveL 7513 to (492.88, 448.08, 132) mm, rotated rx 180 ry 0 rz 160 deg; joints [-0.384, 55.974, 2.288, -157.263, 60.297, 168.269]
  Set speed (16.4 mm/s)
  Call Extruder(13.22166)
  MoveL 7514 to (494.81, 447.85, 132) mm, rotated rx 180 ry 0 rz 160 deg; joints [-0.412, 56.269, 1.691, -157.227, 60.013, 168.15]
  Set speed (16.4 mm/s)
  Call Extruder(19.94142)
  MoveL 7515 to (496.75, 447.7, 132) mm, rotated rx 180 ry 0 rz 160 deg; joints [-0.43, 56.568, 1.087, -157.179, 59.727, 168.024]
  Set speed (16.4 mm/s)
  Call Extruder(26.76534)
  MoveL 7516 to (498.73, 447.61, 132) mm, rotated rx -180 ry 0 rz 160 deg; joints [-0.439, 56.875, 0.467, -157.118, 59.437, 167.888]
  Set speed (16.4 mm/s)
  Call Extruder(33.33010)
  MoveL 7517 to (500.63, 447.6, 132) mm, rotated rx -180 ry 0 rz 160 deg; joints [-0.438, 57.173, -0.134, -157.048, 59.158, 167.75]
  Call Extruder(40.06326)
  MoveL 7518 to (502.59, 447.66, 132) mm, rotated rx 180 ry 0 rz 160 deg; joints [-0.429, 57.48, -0.754, -156.963, 58.872, 167.602]
  Call Extruder(46.61477)
  MoveL 7519 to (504.49, 447.79, 132) mm, rotated rx -180 ry 0 rz 160 deg; joints [-0.411, 57.781, -1.361, -156.87, 58.595, 167.452]
  Set speed (16.4 mm/s)
  Call Extruder(53.34683)
  MoveL 7520 to (506.43, 447.99, 132) mm, rotated rx -180 ry 0 rz 160 deg; joints [-0.384, 58.092, -1.986, -156.763, 58.312, 167.29]
  Set speed (16.4 mm/s)
  Call Extruder(59.90366)
  MoveL 7521 to (508.31, 448.26, 132) mm, rotated rx -180 ry 0 rz 160 deg; joints [-0.349, 58.395, -2.596, -156.647, 58.038, 167.126]
  Set speed (16.4 mm/s)
  Call Extruder(66.53430)
  MoveL 7522 to (510.21, 448.6, 132) mm, rotated rx 180 ry 0 rz 160 deg; joints [-0.305, 58.702, -3.213, -156.52, 57.763, 166.954]
  Set speed (16.4 mm/s)
  Call Extruder(72.62259)
  MoveL 7523 to (511.93, 448.97, 132) mm, rotated rx 180 ry 0 rz 160 deg; joints [-0.258, 58.985, -3.78, -156.393, 57.513, 166.79]
  Call Extruder(79.77258)
  MoveL 7524 to (513.94, 449.48, 132) mm, rotated rx 180 ry 0 rz 160 deg; joints [-0.193, 59.316, -4.445, -156.233, 57.223, 166.591]
  Set speed (16.4 mm/s)
  Call Extruder(86.49314)
  MoveL 7525 to (515.81, 450.04, 132) mm, rotated rx 180 ry 0 rz 160 deg; joints [-0.124, 59.627, -5.069, -156.071, 56.953, 166.397]
  Set speed (16.4 mm/s)
  Call Extruder(93.23424)
  MoveL 7526 to (517.67, 450.66, 132) mm, rotated rx -180 ry 0 rz 160 deg; joints [-0.046, 59.939, -5.692, -155.898, 56.686, 166.196]
  Call Extruder(99.78000)
  MoveL 7527 to (519.44, 451.34, 132) mm, rotated rx -180 ry 0 rz 160 deg; joints [0.036, 60.239, -6.294, -155.721, 56.431, 165.995]
  Set speed (16.4 mm/s)
  Call Extruder(106.48185)
  MoveL 7528 to (521.24, 452.09, 132) mm, rotated rx -180 ry 0 rz 160 deg; joints [0.128, 60.546, -6.906, -155.53, 56.175, 165.784]
  Set speed (16.4 mm/s)
  Call Extruder(112.23120)
  MoveL 7529 to (522.75, 452.79, 132) mm, rotated rx -180 ry 0 rz 160 deg; joints [0.212, 60.807, -7.428, -155.358, 55.959, 165.599]
  Set speed (16.4 mm/s)
  Call Extruder(119.74201)
  MoveL 7530 to (524.69, 453.78, 132) mm, rotated rx -180 ry 0 rz 160 deg; joints [0.33, 61.144, -8.102, -155.124, 55.683, 165.35]
  Set speed (16.4 mm/s)
  Call Extruder(126.48384)
  MoveL 7531 to (526.4, 454.73, 132) mm, rotated rx 180 ry 0 rz 160 deg; joints [0.444, 61.444, -8.7, -154.904, 55.442, 165.122]
  Set speed (16.4 mm/s)
  Call Extruder(133.03931)
  MoveL 7532 to (528.03, 455.72, 132) mm, rotated rx 180 ry 0 rz 160 deg; joints [0.561, 61.733, -9.276, -154.682, 55.212, 164.895]
  Call Extruder(139.77159)
  MoveL 7533 to (529.66, 456.79, 132) mm, rotated rx -180 ry 0 rz 160 deg; joints [0.688, 62.025, -9.858, -154.446, 54.984, 164.658]
  Set speed (16.4 mm/s)
  Call Extruder(146.33181)
  MoveL 7534 to (531.21, 457.9, 132) mm, rotated rx -180 ry 0 rz 160 deg; joints [0.818, 62.306, -10.417, -154.209, 54.768, 164.423]
  Set speed (16.4 mm/s)
  Call Extruder(152.84767)
  MoveL 7535 to (532.71, 459.05, 132) mm, rotated rx -180 ry 0 rz 160 deg; joints [0.952, 62.58, -10.962, -153.966, 54.56, 164.186]
  Set speed (16.4 mm/s)
  Call Extruder(159.51352)
  MoveL 7536 to (534.19, 460.29, 132) mm, rotated rx -180 ry 0 rz 160 deg; joints [1.096, 62.855, -11.51, -153.71, 54.355, 163.94]
  Call Extruder(166.37169)
  MoveL 7537 to (535.68, 461.62, 132) mm, rotated rx 180 ry 0 rz 160 deg; joints [1.249, 63.133, -12.062, -153.441, 54.152, 163.683]
  Call Extruder(172.86429)
  MoveL 7538 to (537.03, 462.93, 132) mm, rotated rx 180 ry 0 rz 160 deg; joints [1.4, 63.39, -12.572, -153.18, 53.969, 163.438]
  Set speed (16.4 mm/s)
  Call Extruder(176.57981)
  MoveL 7539 to (537.79, 463.69, 132) mm, rotated rx 180 ry 0 rz 160 deg; joints [1.488, 63.535, -12.859, -153.029, 53.867, 163.297]
  Set speed (16.4 mm/s)
  Call Extruder(180.20030)
  MoveL 7540 to (538.51, 464.46, 132) mm, rotated rx 180 ry 0 rz 160 deg; joints [1.575, 63.674, -13.135, -152.88, 53.77, 163.159]
  Set speed (16.4 mm/s)
  Call Extruder(183.93457)
  MoveL 7541 to (539.24, 465.26, 132) mm, rotated rx -180 ry 0 rz 160 deg; joints [1.667, 63.815, -13.414, -152.724, 53.674, 163.015]
  Set speed (16.4 mm/s)
  Call Extruder(187.68476)
  MoveL 7542 to (539.95, 466.09, 132) mm, rotated rx 180 ry 0 rz 160 deg; joints [1.761, 63.954, -13.69, -152.566, 53.58, 162.871]
  Call Extruder(191.40872)
  MoveL 7543 to (540.64, 466.92, 132) mm, rotated rx -180 ry 0 rz 160 deg; joints [1.856, 64.09, -13.959, -152.408, 53.49, 162.728]
  Call Extruder(195.05281)
  MoveL 7544 to (541.3, 467.74, 132) mm, rotated rx 180 ry 0 rz 160 deg; joints [1.95, 64.22, -14.218, -152.253, 53.404, 162.587]
  Set speed (16.4 mm/s)
  Call Extruder(198.77549)
  MoveL 7545 to (541.96, 468.6, 132) mm, rotated rx 180 ry 0 rz 160 deg; joints [2.047, 64.352, -14.478, -152.092, 53.319, 162.443]
  Set speed (16.4 mm/s)
  Call Extruder(202.41709)
  MoveL 7546 to (542.58, 469.46, 132) mm, rotated rx -180 ry 0 rz 160 deg; joints [2.144, 64.477, -14.726, -151.934, 53.24, 162.302]
  Set speed (16.4 mm/s)
  Call Extruder(206.10238)
  MoveL 7547 to (543.2, 470.33, 132) mm, rotated rx 180 ry 0 rz 160 deg; joints [2.243, 64.602, -14.975, -151.773, 53.162, 162.16]
  Call Extruder(209.04183)
  MoveL 7548 to (543.67, 471.04, 132) mm, rotated rx 180 ry 0 rz 160 deg; joints [2.323, 64.7, -15.168, -151.644, 53.103, 162.046]
  Set speed (16.4 mm/s)
  Call Extruder(213.58422)
  MoveL 7549 to (544.39, 472.15, 132) mm, rotated rx 180 ry 0 rz 160 deg; joints [2.448, 64.847, -15.459, -151.444, 53.014, 161.871]
  Set speed (16.4 mm/s)
  Call Extruder(217.25938)
  MoveL 7550 to (544.95, 473.05, 132) mm, rotated rx -180 ry 0 rz 160 deg; joints [2.55, 64.964, -15.69, -151.281, 52.946, 161.729]
  Set speed (16.4 mm/s)
  Call Extruder(220.89190)
  MoveL 7551 to (545.48, 473.96, 132) mm, rotated rx 180 ry 0 rz 160 deg; joints [2.652, 65.076, -15.911, -151.119, 52.883, 161.589]
  Set speed (16.4 mm/s)
  Call Extruder(226.71085)
  MoveL 7552 to (546.3, 475.44, 132) mm, rotated rx 180 ry 0 rz 160 deg; joints [2.818, 65.25, -16.256, -150.859, 52.786, 161.366]
  Set speed (16.4 mm/s)
  Call Extruder(231.97509)
  MoveL 7553 to (546.99, 476.8, 132) mm, rotated rx 180 ry 0 rz 160 deg; joints [2.971, 65.4, -16.552, -150.623, 52.708, 161.167]
  Set speed (16.4 mm/s)
  Call Extruder(238.46296)
  MoveL 7554 to (547.8, 478.5, 132) mm, rotated rx 180 ry 0 rz 160 deg; joints [3.161, 65.579, -16.905, -150.331, 52.618, 160.921]
  Call Extruder(246.87306)
  MoveL 7555 to (548.74, 480.75, 132) mm, rotated rx 180 ry 0 rz 160 deg; joints [3.413, 65.792, -17.328, -149.952, 52.52, 160.608]
  Set speed (16.4 mm/s)
  Call Extruder(254.05670)
  MoveL 7556 to (549.47, 482.7, 132) mm, rotated rx 180 ry 0 rz 160 deg; joints [3.632, 65.962, -17.662, -149.628, 52.45, 160.345]
  Set speed (16.4 mm/s)
  Call Extruder(257.92190)
  MoveL 7557 to (549.82, 483.76, 132) mm, rotated rx -180 ry 0 rz 160 deg; joints [3.751, 66.047, -17.83, -149.455, 52.419, 160.206]
  Call Extruder(261.61716)
  MoveL 7558 to (550.15, 484.78, 132) mm, rotated rx 180 ry 0 rz 160 deg; joints [3.865, 66.127, -17.988, -149.289, 52.391, 160.074]
  Set speed (16.4 mm/s)
  Call Extruder(268.78408)
  MoveL 7559 to (550.71, 486.78, 132) mm, rotated rx 180 ry 0 rz 160 deg; joints [4.089, 66.269, -18.269, -148.968, 52.349, 159.822]
  Set speed (16.4 mm/s)
  Call Extruder(272.71331)
  MoveL 7560 to (550.98, 487.89, 132) mm, rotated rx -180 ry 0 rz 160 deg; joints [4.213, 66.341, -18.41, -148.794, 52.332, 159.687]
  Set speed (16.4 mm/s)
  Call Extruder(276.26243)
  MoveL 7561 to (551.22, 488.89, 132) mm, rotated rx -180 ry 0 rz 160 deg; joints [4.325, 66.404, -18.534, -148.637, 52.319, 159.565]
  Set speed (16.4 mm/s)
  Call Extruder(283.75482)
  MoveL 7562 to (551.63, 491.03, 132) mm, rotated rx 180 ry 0 rz 160 deg; joints [4.564, 66.522, -18.768, -148.307, 52.304, 159.316]
  Call Extruder(291.14537)
  MoveL 7563 to (551.96, 493.15, 132) mm, rotated rx 180 ry 0 rz 160 deg; joints [4.801, 66.624, -18.969, -147.986, 52.304, 159.078]
  Call Extruder(298.64121)
  MoveL 7564 to (552.2, 495.31, 132) mm, rotated rx 180 ry 0 rz 160 deg; joints [5.044, 66.712, -19.142, -147.664, 52.32, 158.846]
  Set speed (16.4 mm/s)
  Call Extruder(305.91894)
  MoveL 7565 to (552.34, 497.42, 132) mm, rotated rx 180 ry 0 rz 160 deg; joints [5.282, 66.782, -19.28, -147.357, 52.349, 158.629]
  Set speed (16.4 mm/s)
  Call Extruder(313.30412)
  MoveL 7566 to (552.4, 499.56, 132) mm, rotated rx 180 ry 0 rz 160 deg; joints [5.524, 66.836, -19.386, -147.051, 52.393, 158.42]
  Set speed (16.4 mm/s)
  Call Extruder(320.53404)
  MoveL 7567 to (552.38, 501.66, 132) mm, rotated rx 180 ry 0 rz 160 deg; joints [5.761, 66.874, -19.461, -146.757, 52.45, 158.225]
  Set speed (16.4 mm/s)
  Call Extruder(328.05149)
  MoveL 7568 to (552.26, 503.84, 132) mm, rotated rx 180 ry 0 rz 160 deg; joints [6.009, 66.896, -19.505, -146.458, 52.524, 158.033]
  Call Extruder(335.44292)
  MoveL 7569 to (552.06, 505.97, 132) mm, rotated rx -180 ry 0 rz 160 deg; joints [6.253, 66.902, -19.517, -146.171, 52.611, 157.856]
  Set speed (16.4 mm/s)
  Call Extruder(342.92712)
  MoveL 7570 to (551.77, 508.13, 132) mm, rotated rx 180 ry 0 rz 160 deg; joints [6.5, 66.891, -19.495, -145.888, 52.713, 157.689]
  Set speed (16.4 mm/s)
  Call Extruder(350.21060)
  MoveL 7571 to (551.4, 510.21, 132) mm, rotated rx -180 ry 0 rz 160 deg; joints [6.74, 66.865, -19.444, -145.62, 52.825, 157.538]
  Set speed (16.4 mm/s)
  Call Extruder(357.45090)
  MoveL 7572 to (550.95, 512.26, 132) mm, rotated rx -180 ry 0 rz 160 deg; joints [6.977, 66.823, -19.361, -145.362, 52.95, 157.401]
  Set speed (16.4 mm/s)
  Call Extruder(365.14613)
  MoveL 7573 to (550.38, 514.42, 132) mm, rotated rx -180 ry 0 rz 160 deg; joints [7.229, 66.762, -19.24, -145.096, 53.096, 157.269]
  Set speed (16.4 mm/s)
  Call Extruder(372.16347)
  MoveL 7574 to (549.78, 516.37, 132) mm, rotated rx 180 ry 0 rz 160 deg; joints [7.458, 66.69, -19.099, -144.863, 53.241, 157.161]
  Set speed (16.4 mm/s)
  Call Extruder(376.61045)
  MoveL 7575 to (549.36, 517.59, 132) mm, rotated rx 180 ry 0 rz 160 deg; joints [7.602, 66.637, -18.994, -144.72, 53.34, 157.099]
  Call Extruder(379.66072)
  MoveL 7576 to (549.06, 518.42, 132) mm, rotated rx -180 ry 0 rz 160 deg; joints [7.7, 66.598, -18.918, -144.623, 53.409, 157.059]
  Set speed (16.4 mm/s)
  Call Extruder(387.24172)
  MoveL 7577 to (548.25, 520.47, 132) mm, rotated rx 180 ry 0 rz 160 deg; joints [7.944, 66.49, -18.704, -144.39, 53.589, 156.969]
  Set speed (16.4 mm/s)
  Call Extruder(394.37074)
  MoveL 7578 to (547.4, 522.36, 132) mm, rotated rx 180 ry 0 rz 160 deg; joints [8.171, 66.372, -18.472, -144.18, 53.771, 156.898]
  Set speed (16.4 mm/s)
  Call Extruder(398.18555)
  MoveL 7579 to (546.92, 523.35, 132) mm, rotated rx -180 ry 0 rz 160 deg; joints [8.291, 66.304, -18.337, -144.071, 53.872, 156.865]
  Set speed (16.4 mm/s)
  Call Extruder(401.08508)
  MoveL 7580 to (546.53, 524.1, 132) mm, rotated rx -180 ry 0 rz 160 deg; joints [8.382, 66.249, -18.229, -143.99, 53.952, 156.843]
  Set speed (16.4 mm/s)
  Call Extruder(404.77574)
  MoveL 7581 to (546.03, 525.05, 132) mm, rotated rx 180 ry 0 rz 160 deg; joints [8.498, 66.176, -18.086, -143.889, 54.054, 156.817]
  Call Extruder(408.47569)
  MoveL 7582 to (545.51, 525.99, 132) mm, rotated rx 180 ry 0 rz 160 deg; joints [8.613, 66.099, -17.934, -143.79, 54.16, 156.796]
  Call Extruder(413.00132)
  MoveL 7583 to (544.84, 527.12, 132) mm, rotated rx 180 ry 0 rz 160 deg; joints [8.753, 66.001, -17.74, -143.673, 54.292, 156.773]
  Set speed (16.4 mm/s)
  Call Extruder(416.56033)
  MoveL 7584 to (544.3, 528, 132) mm, rotated rx 180 ry 0 rz 160 deg; joints [8.862, 65.92, -17.58, -143.583, 54.399, 156.758]
  Set speed (16.4 mm/s)
  Call Extruder(419.68475)
  MoveL 7585 to (543.81, 528.76, 132) mm, rotated rx 180 ry 0 rz 160 deg; joints [8.957, 65.847, -17.435, -143.506, 54.494, 156.748]
  Set speed (16.4 mm/s)
  Call Extruder(424.02354)
  MoveL 7586 to (543.11, 529.8, 132) mm, rotated rx 180 ry 0 rz 160 deg; joints [9.088, 65.74, -17.224, -143.402, 54.629, 156.739]
  Set speed (16.4 mm/s)
  Call Extruder(427.78484)
  MoveL 7587 to (542.48, 530.7, 132) mm, rotated rx -180 ry 0 rz 160 deg; joints [9.201, 65.644, -17.035, -143.315, 54.749, 156.733]
  Set speed (16.4 mm/s)
  Call Extruder(430.63090)
  MoveL 7588 to (541.99, 531.36, 132) mm, rotated rx 180 ry 0 rz 160 deg; joints [9.285, 65.569, -16.887, -143.251, 54.841, 156.732]
  Call Extruder(435.10548)
  MoveL 7589 to (541.2, 532.39, 132) mm, rotated rx -180 ry 0 rz 160 deg; joints [9.417, 65.447, -16.646, -143.153, 54.988, 156.734]
  Set speed (16.4 mm/s)
  Call Extruder(438.73449)
  MoveL 7590 to (540.54, 533.21, 132) mm, rotated rx -180 ry 0 rz 160 deg; joints [9.523, 65.346, -16.446, -143.075, 55.109, 156.739]
  Set speed (16.4 mm/s)
  Call Extruder(442.43903)
  MoveL 7591 to (539.85, 534.04, 132) mm, rotated rx 180 ry 0 rz 160 deg; joints [9.63, 65.238, -16.233, -142.999, 55.235, 156.747]
  Set speed (16.4 mm/s)
  Call Extruder(446.14399)
  MoveL 7592 to (539.14, 534.85, 132) mm, rotated rx 180 ry 0 rz 160 deg; joints [9.736, 65.128, -16.015, -142.926, 55.363, 156.758]
  Set speed (16.4 mm/s)
  Call Extruder(449.83144)
  MoveL 7593 to (538.42, 535.64, 132) mm, rotated rx -180 ry 0 rz 160 deg; joints [9.841, 65.016, -15.793, -142.855, 55.492, 156.773]
  Set speed (16.4 mm/s)
  Call Extruder(453.75832)
  MoveL 7594 to (537.64, 536.47, 132) mm, rotated rx 180 ry 0 rz 160 deg; joints [9.951, 64.893, -15.549, -142.782, 55.631, 156.792]
  Set speed (16.4 mm/s)
  Call Extruder(457.32207)
  MoveL 7595 to (536.91, 537.2, 132) mm, rotated rx -180 ry 0 rz 160 deg; joints [10.049, 64.778, -15.323, -142.719, 55.759, 156.812]
  Set speed (16.4 mm/s)
  Call Extruder(460.98180)
  MoveL 7596 to (536.15, 537.94, 132) mm, rotated rx -180 ry 0 rz 160 deg; joints [10.149, 64.658, -15.085, -142.656, 55.892, 156.836]
  Set speed (16.4 mm/s)
  Call Extruder(464.60000)
  MoveL 7597 to (535.38, 538.66, 132) mm, rotated rx 180 ry 0 rz 160 deg; joints [10.247, 64.537, -14.845, -142.596, 56.025, 156.862]
  Set speed (16.4 mm/s)
  Call Extruder(467.58760)
  MoveL 7598 to (534.74, 539.24, 132) mm, rotated rx 180 ry 0 rz 160 deg; joints [10.327, 64.435, -14.643, -142.548, 56.136, 156.886]
  Set speed (16.4 mm/s)
  Call Extruder(471.95509)
  MoveL 7599 to (533.78, 540.07, 132) mm, rotated rx 180 ry 0 rz 160 deg; joints [10.442, 64.283, -14.342, -142.481, 56.299, 156.924]
  Set speed (16.4 mm/s)
  Call Extruder(475.70088)
  MoveL 7600 to (532.94, 540.76, 132) mm, rotated rx 180 ry 0 rz 160 deg; joints [10.54, 64.149, -14.077, -142.427, 56.441, 156.96]
  Set speed (16.4 mm/s)
  Call Extruder(479.38729)
  MoveL 7601 to (532.1, 541.43, 132) mm, rotated rx 180 ry 0 rz 160 deg; joints [10.634, 64.016, -13.812, -142.376, 56.582, 156.999]
  Set speed (16.4 mm/s)
  Call Extruder(483.21662)
  MoveL 7602 to (531.21, 542.1, 132) mm, rotated rx -180 ry 0 rz 160 deg; joints [10.73, 63.874, -13.532, -142.326, 56.73, 157.042]
  Set speed (16.4 mm/s)
  Call Extruder(486.78722)
  MoveL 7603 to (530.37, 542.71, 132) mm, rotated rx -180 ry 0 rz 160 deg; joints [10.819, 63.741, -13.268, -142.281, 56.868, 157.085]
  Set speed (16.4 mm/s)
  Call Extruder(490.49059)
  MoveL 7604 to (529.49, 543.32, 132) mm, rotated rx -180 ry 0 rz 160 deg; joints [10.909, 63.6, -12.988, -142.236, 57.013, 157.132]
  Set speed (16.4 mm/s)
  Call Extruder(494.18466)
  MoveL 7605 to (528.6, 543.91, 132) mm, rotated rx -180 ry 0 rz 160 deg; joints [10.998, 63.457, -12.705, -142.195, 57.158, 157.181]
  Set speed (16.4 mm/s)
  Call Extruder(497.97086)
  MoveL 7606 to (527.67, 544.5, 132) mm, rotated rx -180 ry 0 rz 160 deg; joints [11.087, 63.309, -12.411, -142.155, 57.308, 157.235]
  Set speed (16.4 mm/s)
  Call Extruder(501.63543)
  MoveL 7607 to (526.76, 545.05, 132) mm, rotated rx 180 ry 0 rz 160 deg; joints [11.171, 63.164, -12.122, -142.119, 57.454, 157.29]
  Set speed (16.4 mm/s)
  Call Extruder(505.24462)
  MoveL 7608 to (525.86, 545.58, 132) mm, rotated rx -180 ry 0 rz 160 deg; joints [11.253, 63.019, -11.835, -142.085, 57.598, 157.346]
  Set speed (16.4 mm/s)
  Call Extruder(508.96161)
  MoveL 7609 to (524.92, 546.11, 132) mm, rotated rx -180 ry 0 rz 160 deg; joints [11.336, 62.868, -11.535, -142.053, 57.747, 157.406]
  Set speed (16.4 mm/s)
  Call Extruder(512.69366)
  MoveL 7610 to (523.96, 546.61, 132) mm, rotated rx 180 ry 0 rz 160 deg; joints [11.417, 62.714, -11.229, -142.023, 57.898, 157.469]
  Set speed (16.4 mm/s)
  Call Extruder(516.29797)
  MoveL 7611 to (523.02, 547.08, 132) mm, rotated rx 180 ry 0 rz 160 deg; joints [11.494, 62.565, -10.931, -141.996, 58.044, 157.532]
  Set speed (16.4 mm/s)
  Call Extruder(520.16566)
  MoveL 7612 to (522.01, 547.56, 132) mm, rotated rx -180 ry 0 rz 160 deg; joints [11.574, 62.402, -10.608, -141.97, 58.202, 157.602]
  Set speed (16.4 mm/s)
  Call Extruder(523.79434)
  MoveL 7613 to (521.05, 547.99, 132) mm, rotated rx -180 ry 0 rz 160 deg; joints [11.647, 62.248, -10.302, -141.949, 58.35, 157.671]
  Set speed (16.4 mm/s)
  Call Extruder(527.29648)
  MoveL 7614 to (520.11, 548.39, 132) mm, rotated rx -180 ry 0 rz 160 deg; joints [11.717, 62.099, -10.004, -141.93, 58.492, 157.739]
  Set speed (16.4 mm/s)
  Call Extruder(531.17801)
  MoveL 7615 to (519.07, 548.81, 132) mm, rotated rx -180 ry 0 rz 160 deg; joints [11.791, 61.931, -9.67, -141.912, 58.651, 157.817]
  Set speed (16.4 mm/s)
  Call Extruder(535.11597)
  MoveL 7616 to (518, 549.21, 132) mm, rotated rx 180 ry 0 rz 160 deg; joints [11.865, 61.76, -9.33, -141.895, 58.813, 157.898]
  Set speed (16.4 mm/s)
  Call Extruder(542.12999)
  MoveL 7617 to (516.08, 549.88, 132) mm, rotated rx -180 ry 0 rz 160 deg; joints [11.991, 61.452, -8.715, -141.873, 59.101, 158.048]
  Call Extruder(549.57189)
  MoveL 7618 to (514.01, 550.5, 132) mm, rotated rx 180 ry 0 rz 160 deg; joints [12.116, 61.121, -8.054, -141.858, 59.407, 158.216]
  Call Extruder(556.88355)
  MoveL 7619 to (511.95, 551.02, 132) mm, rotated rx 180 ry 0 rz 160 deg; joints [12.231, 60.791, -7.397, -141.854, 59.707, 158.388]
  Set speed (16.4 mm/s)
  Call Extruder(564.43861)
  MoveL 7620 to (509.81, 551.48, 132) mm, rotated rx 180 ry 0 rz 160 deg; joints [12.34, 60.448, -6.711, -141.859, 60.017, 158.574]
  Set speed (16.4 mm/s)
  Call Extruder(571.88900)
  MoveL 7621 to (507.68, 551.84, 132) mm, rotated rx 180 ry 0 rz 160 deg; joints [12.439, 60.107, -6.029, -141.874, 60.321, 158.764]
  Set speed (16.4 mm/s)
  Call Extruder(579.18834)
  MoveL 7622 to (505.58, 552.11, 132) mm, rotated rx 180 ry 0 rz 160 deg; joints [12.527, 59.771, -5.356, -141.897, 60.618, 158.956]
  Set speed (16.4 mm/s)
  Call Extruder(586.61525)
  MoveL 7623 to (503.43, 552.29, 132) mm, rotated rx 180 ry 0 rz 160 deg; joints [12.607, 59.427, -4.668, -141.931, 60.918, 159.158]
  Call Extruder(594.06689)
  MoveL 7624 to (501.27, 552.39, 132) mm, rotated rx 180 ry 0 rz 160 deg; joints [12.677, 59.082, -3.975, -141.974, 61.216, 159.366]
  Set speed (16.4 mm/s)
  Call Extruder(601.34725)
  MoveL 7625 to (499.15, 552.4, 132) mm, rotated rx 180 ry 0 rz 160 deg; joints [12.736, 58.744, -3.297, -142.025, 61.505, 159.575]
  Set speed (10.0 mm/s)
  MoveL 7626 to (499.15, 552.4, 136) mm, rotated rx -180 ry 0 rz 160 deg; joints [12.736, 58.15, -3.106, -141.89, 61.188, 159.292]
  Set speed (120.0 mm/s)
  MoveL 7627 to (499.19, 550.62, 136) mm, rotated rx 180 ry 0 rz 160 deg; joints [12.518, 58.091, -2.988, -142.142, 61.157, 159.445]
  Set speed (16.5 mm/s)
  Call Extruder(608.49649)
  MoveL 7628 to (497.1, 550.54, 136) mm, rotated rx 180 ry 0 rz 160 deg; joints [12.566, 57.755, -2.318, -142.204, 61.438, 159.655]
  Set speed (16.5 mm/s)
  Call Extruder(615.60646)
  MoveL 7629 to (495.03, 550.38, 136) mm, rotated rx 180 ry 0 rz 160 deg; joints [12.602, 57.422, -1.653, -142.275, 61.713, 159.868]
  Set speed (16.5 mm/s)
  Call Extruder(622.62998)
  MoveL 7630 to (492.99, 550.13, 136) mm, rotated rx -180 ry 0 rz 160 deg; joints [12.629, 57.094, -0.997, -142.354, 61.982, 160.082]
  Call Extruder(629.67638)
  MoveL 7631 to (490.95, 549.81, 136) mm, rotated rx 180 ry 0 rz 160 deg; joints [12.645, 56.767, -0.342, -142.443, 62.247, 160.3]
  Set speed (16.5 mm/s)
  Call Extruder(636.89614)
  MoveL 7632 to (488.88, 549.39, 136) mm, rotated rx -180 ry 0 rz 160 deg; joints [12.65, 56.434, 0.326, -142.544, 62.514, 160.527]
  Set speed (16.5 mm/s)
  Call Extruder(643.81200)
  MoveL 7633 to (486.92, 548.91, 136) mm, rotated rx 180 ry 0 rz 160 deg; joints [12.645, 56.118, 0.96, -142.649, 62.765, 160.747]
  Call Extruder(650.79161)
  MoveL 7634 to (484.96, 548.34, 136) mm, rotated rx -180 ry 0 rz 160 deg; joints [12.629, 55.801, 1.595, -142.765, 63.013, 160.972]
  Set speed (16.5 mm/s)
  Call Extruder(654.50056)
  MoveL 7635 to (483.93, 548, 136) mm, rotated rx -180 ry 0 rz 160 deg; joints [12.615, 55.635, 1.929, -142.831, 63.142, 161.092]
  Set speed (16.5 mm/s)
  Call Extruder(658.00438)
  MoveL 7636 to (482.97, 547.67, 136) mm, rotated rx 180 ry 0 rz 160 deg; joints [12.601, 55.478, 2.243, -142.894, 63.263, 161.205]
  Call Extruder(661.66539)
  MoveL 7637 to (481.97, 547.3, 136) mm, rotated rx 180 ry 0 rz 160 deg; joints [12.582, 55.316, 2.57, -142.964, 63.388, 161.325]
  Call Extruder(665.64946)
  MoveL 7638 to (480.88, 546.88, 136) mm, rotated rx -180 ry 0 rz 160 deg; joints [12.559, 55.14, 2.923, -143.041, 63.522, 161.455]
  Set speed (16.5 mm/s)
  Call Extruder(673.72577)
  MoveL 7639 to (478.71, 545.94, 136) mm, rotated rx 180 ry 0 rz 160 deg; joints [12.501, 54.788, 3.631, -143.209, 63.789, 161.721]
  Set speed (16.5 mm/s)
  Call Extruder(680.88720)
  MoveL 7640 to (476.84, 545.02, 136) mm, rotated rx 180 ry 0 rz 160 deg; joints [12.437, 54.482, 4.247, -143.368, 64.018, 161.958]
  Set speed (16.5 mm/s)
  Call Extruder(686.31548)
  MoveL 7641 to (475.44, 544.27, 136) mm, rotated rx -180 ry 0 rz 160 deg; joints [12.38, 54.254, 4.707, -143.495, 64.186, 162.137]
  Set speed (16.5 mm/s)
  Call Extruder(689.85646)
  MoveL 7642 to (474.54, 543.75, 136) mm, rotated rx -180 ry 0 rz 160 deg; joints [12.339, 54.107, 5.004, -143.581, 64.294, 162.255]
  Call Extruder(693.54916)
  MoveL 7643 to (473.61, 543.2, 136) mm, rotated rx -180 ry 0 rz 160 deg; joints [12.294, 53.955, 5.31, -143.673, 64.405, 162.377]
  Call Extruder(696.91434)
  MoveL 7644 to (472.78, 542.68, 136) mm, rotated rx -180 ry 0 rz 160 deg; joints [12.25, 53.818, 5.587, -143.759, 64.504, 162.489]
  Set speed (16.5 mm/s)
  Call Extruder(700.51041)
  MoveL 7645 to (471.9, 542.1, 136) mm, rotated rx 180 ry 0 rz 160 deg; joints [12.2, 53.673, 5.879, -143.853, 64.608, 162.608]
  Set speed (16.5 mm/s)
  Call Extruder(704.10624)
  MoveL 7646 to (471.03, 541.51, 136) mm, rotated rx -180 ry 0 rz 160 deg; joints [12.147, 53.53, 6.169, -143.949, 64.71, 162.727]
  Set speed (16.5 mm/s)
  Call Extruder(707.61168)
  MoveL 7647 to (470.19, 540.92, 136) mm, rotated rx 180 ry 0 rz 160 deg; joints [12.093, 53.392, 6.447, -144.046, 64.808, 162.843]
  Set speed (16.5 mm/s)
  Call Extruder(711.13337)
  MoveL 7648 to (469.37, 540.3, 136) mm, rotated rx 180 ry 0 rz 160 deg; joints [12.036, 53.255, 6.723, -144.145, 64.904, 162.959]
  Call Extruder(714.65068)
  MoveL 7649 to (468.56, 539.67, 136) mm, rotated rx 180 ry 0 rz 160 deg; joints [11.976, 53.12, 6.996, -144.246, 64.999, 163.075]
  Set speed (16.5 mm/s)
  Call Extruder(718.21663)
  MoveL 7650 to (467.75, 539.01, 136) mm, rotated rx -180 ry 0 rz 160 deg; joints [11.912, 52.986, 7.268, -144.35, 65.092, 163.192]
  Set speed (16.5 mm/s)
  Call Extruder(721.89471)
  MoveL 7651 to (466.92, 538.32, 136) mm, rotated rx 180 ry 0 rz 160 deg; joints [11.843, 52.849, 7.546, -144.461, 65.186, 163.312]
  Call Extruder(725.34597)
  MoveL 7652 to (466.17, 537.65, 136) mm, rotated rx 180 ry 0 rz 160 deg; joints [11.776, 52.722, 7.802, -144.566, 65.273, 163.425]
  Set speed (16.5 mm/s)
  Call Extruder(728.97311)
  MoveL 7653 to (465.39, 536.94, 136) mm, rotated rx 180 ry 0 rz 160 deg; joints [11.703, 52.592, 8.067, -144.679, 65.361, 163.543]
  Set speed (16.5 mm/s)
  Call Extruder(732.49599)
  MoveL 7654 to (464.64, 536.23, 136) mm, rotated rx -180 ry 0 rz 160 deg; joints [11.629, 52.466, 8.321, -144.791, 65.445, 163.657]
  Set speed (16.5 mm/s)
  Call Extruder(735.94730)
  MoveL 7655 to (463.93, 535.52, 136) mm, rotated rx 180 ry 0 rz 160 deg; joints [11.554, 52.346, 8.565, -144.903, 65.526, 163.768]
  Set speed (16.5 mm/s)
  Call Extruder(739.45782)
  MoveL 7656 to (463.21, 534.78, 136) mm, rotated rx 180 ry 0 rz 160 deg; joints [11.475, 52.225, 8.81, -145.019, 65.605, 163.881]
  Set speed (16.5 mm/s)
  Call Extruder(743.01106)
  MoveL 7657 to (462.51, 534.01, 136) mm, rotated rx -180 ry 0 rz 160 deg; joints [11.392, 52.105, 9.053, -145.138, 65.683, 163.994]
  Set speed (16.5 mm/s)
  Call Extruder(746.54539)
  MoveL 7658 to (461.82, 533.24, 136) mm, rotated rx -180 ry 0 rz 160 deg; joints [11.307, 51.988, 9.291, -145.259, 65.759, 164.106]
  Set speed (16.5 mm/s)
  Call Extruder(752.24420)
  MoveL 7659 to (460.75, 531.97, 136) mm, rotated rx 180 ry 0 rz 160 deg; joints [11.165, 51.804, 9.665, -145.457, 65.877, 164.286]
  Set speed (16.5 mm/s)
  Call Extruder(757.13737)
  MoveL 7660 to (459.86, 530.84, 136) mm, rotated rx 180 ry 0 rz 160 deg; joints [11.037, 51.651, 9.976, -145.632, 65.972, 164.439]
  Set speed (16.5 mm/s)
  Call Extruder(760.73702)
  MoveL 7661 to (459.23, 530, 136) mm, rotated rx -180 ry 0 rz 160 deg; joints [10.94, 51.541, 10.199, -145.763, 66.04, 164.551]
  Set speed (16.5 mm/s)
  Call Extruder(765.04950)
  MoveL 7662 to (458.49, 528.98, 136) mm, rotated rx 180 ry 0 rz 160 deg; joints [10.82, 51.413, 10.459, -145.922, 66.118, 164.683]
  Set speed (16.5 mm/s)
  Call Extruder(770.53662)
  MoveL 7663 to (457.6, 527.65, 136) mm, rotated rx 180 ry 0 rz 160 deg; joints [10.663, 51.255, 10.78, -146.128, 66.212, 164.85]
  Set speed (16.5 mm/s)
  Call Extruder(774.84410)
  MoveL 7664 to (456.92, 526.59, 136) mm, rotated rx -180 ry 0 rz 160 deg; joints [10.535, 51.136, 11.024, -146.293, 66.281, 164.979]
  Set speed (16.5 mm/s)
  Call Extruder(778.53143)
  MoveL 7665 to (456.36, 525.66, 136) mm, rotated rx 180 ry 0 rz 160 deg; joints [10.423, 51.036, 11.226, -146.436, 66.338, 165.089]
  Set speed (16.5 mm/s)
  Call Extruder(781.99604)
  MoveL 7666 to (455.86, 524.78, 136) mm, rotated rx 180 ry 0 rz 160 deg; joints [10.316, 50.946, 11.41, -146.573, 66.389, 165.191]
  Set speed (16.5 mm/s)
  Call Extruder(785.51785)
  MoveL 7667 to (455.37, 523.88, 136) mm, rotated rx -180 ry 0 rz 160 deg; joints [10.204, 50.856, 11.593, -146.712, 66.438, 165.294]
  Call Extruder(789.04679)
  MoveL 7668 to (454.89, 522.97, 136) mm, rotated rx -180 ry 0 rz 160 deg; joints [10.091, 50.769, 11.77, -146.854, 66.485, 165.396]
  Set speed (16.5 mm/s)
  Call Extruder(792.62530)
  MoveL 7669 to (454.42, 522.03, 136) mm, rotated rx 180 ry 0 rz 160 deg; joints [9.973, 50.684, 11.945, -146.999, 66.53, 165.498]
  Set speed (16.5 mm/s)
  Call Extruder(796.25901)
  MoveL 7670 to (453.98, 521.07, 136) mm, rotated rx 180 ry 0 rz 160 deg; joints [9.851, 50.6, 12.115, -147.148, 66.572, 165.601]
  Call Extruder(799.80217)
  MoveL 7671 to (453.55, 520.13, 136) mm, rotated rx 180 ry 0 rz 160 deg; joints [9.731, 50.521, 12.277, -147.294, 66.612, 165.7]
  Set speed (16.5 mm/s)
  Call Extruder(806.77120)
  MoveL 7672 to (452.78, 518.24, 136) mm, rotated rx 180 ry 0 rz 160 deg; joints [9.488, 50.374, 12.577, -147.586, 66.681, 165.891]
  Set speed (16.5 mm/s)
  Call Extruder(810.42356)
  MoveL 7673 to (452.41, 517.24, 136) mm, rotated rx 180 ry 0 rz 160 deg; joints [9.358, 50.301, 12.725, -147.741, 66.713, 165.99]
  Call Extruder(813.79848)
  MoveL 7674 to (452.08, 516.31, 136) mm, rotated rx -180 ry 0 rz 160 deg; joints [9.237, 50.236, 12.857, -147.885, 66.741, 166.08]
  Set speed (16.5 mm/s)
  Call Extruder(820.81142)
  MoveL 7675 to (451.46, 514.36, 136) mm, rotated rx -180 ry 0 rz 160 deg; joints [8.978, 50.111, 13.114, -148.188, 66.791, 166.263]
  Set speed (16.5 mm/s)
  Call Extruder(825.29508)
  MoveL 7676 to (451.11, 513.1, 136) mm, rotated rx -180 ry 0 rz 160 deg; joints [8.81, 50.037, 13.265, -148.383, 66.816, 166.377]
  Set speed (16.5 mm/s)
  Call Extruder(828.81982)
  MoveL 7677 to (450.85, 512.1, 136) mm, rotated rx 180 ry 0 rz 160 deg; joints [8.676, 49.982, 13.378, -148.537, 66.834, 166.465]
  Set speed (16.5 mm/s)
  Call Extruder(835.11832)
  MoveL 7678 to (450.44, 510.31, 136) mm, rotated rx 180 ry 0 rz 160 deg; joints [8.433, 49.891, 13.564, -148.815, 66.859, 166.62]
  Set speed (16.5 mm/s)
  Call Extruder(842.33801)
  MoveL 7679 to (450.05, 508.23, 136) mm, rotated rx -180 ry 0 rz 160 deg; joints [8.15, 49.799, 13.752, -149.136, 66.876, 166.792]
  Set speed (16.5 mm/s)
  Call Extruder(849.41607)
  MoveL 7680 to (449.76, 506.18, 136) mm, rotated rx 180 ry 0 rz 160 deg; joints [7.867, 49.721, 13.911, -149.453, 66.882, 166.954]
  Set speed (16.5 mm/s)
  Call Extruder(856.50118)
  MoveL 7681 to (449.55, 504.12, 136) mm, rotated rx -180 ry 0 rz 160 deg; joints [7.581, 49.656, 14.045, -149.772, 66.877, 167.111]
  Set speed (16.5 mm/s)
  Call Extruder(863.48865)
  MoveL 7682 to (449.42, 502.08, 136) mm, rotated rx -180 ry 0 rz 160 deg; joints [7.295, 49.603, 14.152, -150.086, 66.861, 167.26]
  Call Extruder(871.03894)
  MoveL 7683 to (449.38, 499.88, 136) mm, rotated rx 180 ry 0 rz 160 deg; joints [6.984, 49.561, 14.239, -150.426, 66.831, 167.414]
  Set speed (16.5 mm/s)
  Call Extruder(877.02478)
  MoveL 7684 to (449.41, 498.13, 136) mm, rotated rx 180 ry 0 rz 160 deg; joints [6.735, 49.537, 14.287, -150.695, 66.799, 167.531]
  Call Extruder(883.24429)
  MoveL 7685 to (449.51, 496.31, 136) mm, rotated rx 180 ry 0 rz 160 deg; joints [6.476, 49.523, 14.317, -150.974, 66.756, 167.648]
  Set speed (16.5 mm/s)
  Call Extruder(889.70043)
  MoveL 7686 to (449.68, 494.43, 136) mm, rotated rx 180 ry 0 rz 160 deg; joints [6.207, 49.518, 14.328, -151.262, 66.704, 167.764]
  Call Extruder(896.06271)
  MoveL 7687 to (449.92, 492.59, 136) mm, rotated rx 180 ry 0 rz 160 deg; joints [5.941, 49.523, 14.316, -151.543, 66.642, 167.873]
  Set speed (16.5 mm/s)
  Call Extruder(902.52307)
  MoveL 7688 to (450.23, 490.73, 136) mm, rotated rx 180 ry 0 rz 160 deg; joints [5.672, 49.54, 14.283, -151.826, 66.571, 167.978]
  Set speed (16.5 mm/s)
  Call Extruder(908.73828)
  MoveL 7689 to (450.6, 488.94, 136) mm, rotated rx 180 ry 0 rz 160 deg; joints [5.415, 49.566, 14.229, -152.095, 66.494, 168.073]
  Set speed (16.5 mm/s)
  Call Extruder(915.19741)
  MoveL 7690 to (451.05, 487.11, 136) mm, rotated rx 180 ry 0 rz 160 deg; joints [5.148, 49.602, 14.154, -152.372, 66.405, 168.167]
  Set speed (16.5 mm/s)
  Call Extruder(921.48062)
  MoveL 7691 to (451.55, 485.34, 136) mm, rotated rx -180 ry 0 rz 160 deg; joints [4.891, 49.649, 14.059, -152.637, 66.309, 168.253]
  Call Extruder(927.86148)
  MoveL 7692 to (452.12, 483.57, 136) mm, rotated rx -180 ry 0 rz 160 deg; joints [4.632, 49.706, 13.942, -152.901, 66.203, 168.334]
  Call Extruder(934.40907)
  MoveL 7693 to (452.78, 481.77, 136) mm, rotated rx -180 ry 0 rz 160 deg; joints [4.37, 49.775, 13.801, -153.168, 66.086, 168.412]
  Call Extruder(940.78790)
  MoveL 7694 to (453.48, 480.04, 136) mm, rotated rx -180 ry 0 rz 160 deg; joints [4.118, 49.852, 13.642, -153.422, 65.963, 168.482]
  Set speed (16.5 mm/s)
  Call Extruder(946.96403)
  MoveL 7695 to (454.22, 478.4, 136) mm, rotated rx -180 ry 0 rz 160 deg; joints [3.878, 49.937, 13.47, -153.662, 65.836, 168.544]
  Call Extruder(953.53420)
  MoveL 7696 to (455.07, 476.68, 136) mm, rotated rx -180 ry 0 rz 160 deg; joints [3.627, 50.037, 13.265, -153.911, 65.693, 168.604]
  Set speed (16.5 mm/s)
  Call Extruder(959.86334)
  MoveL 7697 to (455.95, 475.05, 136) mm, rotated rx -180 ry 0 rz 160 deg; joints [3.39, 50.143, 13.048, -154.144, 65.547, 168.657]
  Call Extruder(966.17455)
  MoveL 7698 to (456.89, 473.46, 136) mm, rotated rx 180 ry 0 rz 160 deg; joints [3.159, 50.258, 12.813, -154.369, 65.393, 168.702]
  Set speed (16.5 mm/s)
  Call Extruder(972.56656)
  MoveL 7699 to (457.9, 471.89, 136) mm, rotated rx 180 ry 0 rz 160 deg; joints [2.931, 50.384, 12.555, -154.59, 65.23, 168.743]
  Set speed (16.5 mm/s)
  Call Extruder(978.94047)
  MoveL 7700 to (458.97, 470.36, 136) mm, rotated rx 180 ry 0 rz 160 deg; joints [2.709, 50.52, 12.279, -154.802, 65.059, 168.778]
  Set speed (16.5 mm/s)
  Call Extruder(985.32155)
  MoveL 7701 to (460.09, 468.87, 136) mm, rotated rx 180 ry 0 rz 160 deg; joints [2.493, 50.664, 11.985, -155.006, 64.881, 168.806]
  Set speed (16.5 mm/s)
  Call Extruder(991.73146)
  MoveL 7702 to (461.27, 467.41, 136) mm, rotated rx 180 ry 0 rz 160 deg; joints [2.283, 50.818, 11.671, -155.202, 64.696, 168.829]
  Set speed (16.5 mm/s)
  Call Extruder(998.09863)
  MoveL 7703 to (462.49, 466.01, 136) mm, rotated rx -180 ry 0 rz 160 deg; joints [2.081, 50.98, 11.341, -155.387, 64.504, 168.845]
  Set speed (16.5 mm/s)
  Call Extruder(1004.53743)
  MoveL 7704 to (463.78, 464.64, 136) mm, rotated rx -180 ry 0 rz 160 deg; joints [1.885, 51.152, 10.99, -155.566, 64.303, 168.855]
  Set speed (16.5 mm/s)
  Call Extruder(1010.67345)
  MoveL 7705 to (465.06, 463.37, 136) mm, rotated rx -180 ry 0 rz 160 deg; joints [1.705, 51.324, 10.64, -155.726, 64.106, 168.859]
  Call Extruder(1017.18778)
  MoveL 7706 to (466.46, 462.09, 136) mm, rotated rx -180 ry 0 rz 160 deg; joints [1.522, 51.515, 10.251, -155.887, 63.891, 168.857]
  Set speed (16.5 mm/s)
  Call Extruder(1023.64500)
  MoveL 7707 to (467.9, 460.86, 136) mm, rotated rx -180 ry 0 rz 160 deg; joints [1.348, 51.713, 9.85, -156.036, 63.671, 168.848]
  Call Extruder(1029.90947)
  MoveL 7708 to (469.33, 459.73, 136) mm, rotated rx -180 ry 0 rz 160 deg; joints [1.188, 51.912, 9.445, -156.169, 63.452, 168.833]
  Set speed (16.5 mm/s)
  Call Extruder(1035.89590)
  MoveL 7709 to (470.74, 458.69, 136) mm, rotated rx 180 ry 0 rz 160 deg; joints [1.043, 52.109, 9.046, -156.288, 63.239, 168.813]
  Call Extruder(1042.67978)
  MoveL 7710 to (472.38, 457.58, 136) mm, rotated rx 180 ry 0 rz 160 deg; joints [0.888, 52.34, 8.577, -156.41, 62.991, 168.783]
  Set speed (16.5 mm/s)
  Call Extruder(1049.14552)
  MoveL 7711 to (473.99, 456.58, 136) mm, rotated rx 180 ry 0 rz 160 deg; joints [0.749, 52.567, 8.116, -156.515, 62.75, 168.748]
  Set speed (16.5 mm/s)
  Call Extruder(1055.53163)
  MoveL 7712 to (475.6, 455.65, 136) mm, rotated rx 180 ry 0 rz 160 deg; joints [0.621, 52.798, 7.648, -156.608, 62.507, 168.707]
  Set speed (16.5 mm/s)
  Call Extruder(1061.85243)
  MoveL 7713 to (477.24, 454.78, 136) mm, rotated rx -180 ry 0 rz 160 deg; joints [0.503, 53.034, 7.172, -156.689, 62.263, 168.66]
  Set speed (16.5 mm/s)
  Call Extruder(1068.11711)
  MoveL 7714 to (478.89, 453.99, 136) mm, rotated rx -180 ry 0 rz 160 deg; joints [0.394, 53.273, 6.688, -156.758, 62.017, 168.607]
  Set speed (16.5 mm/s)
  Call Extruder(1074.37624)
  MoveL 7715 to (480.57, 453.26, 136) mm, rotated rx -180 ry 0 rz 160 deg; joints [0.295, 53.517, 6.193, -156.815, 61.767, 168.547]
  Set speed (16.5 mm/s)
  Call Extruder(1080.86915)
  MoveL 7716 to (482.33, 452.56, 136) mm, rotated rx 180 ry 0 rz 160 deg; joints [0.202, 53.777, 5.67, -156.863, 61.506, 168.478]
  Set speed (16.5 mm/s)
  Call Extruder(1087.39904)
  MoveL 7717 to (484.13, 451.93, 136) mm, rotated rx 180 ry 0 rz 160 deg; joints [0.117, 54.043, 5.133, -156.9, 61.24, 168.402]
  Call Extruder(1093.63621)
  MoveL 7718 to (485.87, 451.39, 136) mm, rotated rx 180 ry 0 rz 160 deg; joints [0.046, 54.302, 4.61, -156.923, 60.983, 168.323]
  Call Extruder(1100.07179)
  MoveL 7719 to (487.69, 450.9, 136) mm, rotated rx 180 ry 0 rz 160 deg; joints [-0.019, 54.574, 4.062, -156.935, 60.716, 168.234]
  Set speed (16.5 mm/s)
  Call Extruder(1106.27321)
  MoveL 7720 to (489.45, 450.49, 136) mm, rotated rx -180 ry 0 rz 160 deg; joints [-0.072, 54.841, 3.526, -156.935, 60.457, 168.142]
  Set speed (16.5 mm/s)
  Call Extruder(1112.74464)
  MoveL 7721 to (491.31, 450.13, 136) mm, rotated rx -180 ry 0 rz 160 deg; joints [-0.119, 55.123, 2.958, -156.924, 60.184, 168.039]
  Set speed (16.5 mm/s)
  Call Extruder(1118.86340)
  MoveL 7722 to (493.08, 449.85, 136) mm, rotated rx -180 ry 0 rz 160 deg; joints [-0.154, 55.393, 2.415, -156.902, 59.926, 167.936]
  Set speed (16.5 mm/s)
  Call Extruder(1125.58091)
  MoveL 7723 to (495.03, 449.62, 136) mm, rotated rx 180 ry 0 rz 160 deg; joints [-0.183, 55.693, 1.812, -156.866, 59.641, 167.815]
  Set speed (16.5 mm/s)
  Call Extruder(1131.85927)
  MoveL 7724 to (496.86, 449.48, 136) mm, rotated rx 180 ry 0 rz 160 deg; joints [-0.201, 55.976, 1.243, -156.82, 59.375, 167.695]
  Set speed (16.5 mm/s)
  Call Extruder(1138.41084)
  MoveL 7725 to (498.77, 449.39, 136) mm, rotated rx 180 ry 0 rz 160 deg; joints [-0.211, 56.275, 0.644, -156.761, 59.097, 167.563]
  Set speed (16.5 mm/s)
  Call Extruder(1144.70555)
  MoveL 7726 to (500.61, 449.38, 136) mm, rotated rx 180 ry 0 rz 160 deg; joints [-0.211, 56.565, 0.064, -156.692, 58.83, 167.429]
  Call Extruder(1151.16030)
  MoveL 7727 to (502.5, 449.44, 136) mm, rotated rx 180 ry 0 rz 160 deg; joints [-0.203, 56.863, -0.534, -156.611, 58.557, 167.285]
  Set speed (16.5 mm/s)
  Call Extruder(1157.45323)
  MoveL 7728 to (504.33, 449.56, 136) mm, rotated rx 180 ry 0 rz 160 deg; joints [-0.187, 57.156, -1.12, -156.52, 58.291, 167.139]
  Set speed (16.5 mm/s)
  Call Extruder(1163.90773)
  MoveL 7729 to (506.21, 449.76, 136) mm, rotated rx 180 ry 0 rz 160 deg; joints [-0.161, 57.458, -1.723, -156.416, 58.021, 166.981]
  Set speed (16.5 mm/s)
  Call Extruder(1170.08270)
  MoveL 7730 to (508, 450.01, 136) mm, rotated rx 180 ry 0 rz 160 deg; joints [-0.129, 57.747, -2.301, -156.306, 57.763, 166.825]
  Set speed (16.5 mm/s)
  Call Extruder(1176.58859)
  MoveL 7731 to (509.87, 450.35, 136) mm, rotated rx -180 ry 0 rz 160 deg; joints [-0.086, 58.052, -2.911, -156.179, 57.495, 166.654]
  Set speed (16.5 mm/s)
  Call Extruder(1182.35011)
  MoveL 7732 to (511.52, 450.71, 136) mm, rotated rx -180 ry 0 rz 160 deg; joints [-0.042, 58.323, -3.451, -156.058, 57.259, 166.497]
  Call Extruder(1189.23561)
  MoveL 7733 to (513.47, 451.2, 136) mm, rotated rx 180 ry 0 rz 160 deg; joints [0.02, 58.646, -4.095, -155.902, 56.98, 166.302]
  Set speed (16.5 mm/s)
  Call Extruder(1195.69763)
  MoveL 7734 to (515.28, 451.74, 136) mm, rotated rx 180 ry 0 rz 160 deg; joints [0.086, 58.948, -4.698, -155.746, 56.722, 166.114]
  Call Extruder(1202.14623)
  MoveL 7735 to (517.07, 452.34, 136) mm, rotated rx 180 ry 0 rz 160 deg; joints [0.16, 59.249, -5.296, -155.578, 56.468, 165.919]
  Call Extruder(1208.43742)
  MoveL 7736 to (518.79, 452.99, 136) mm, rotated rx 180 ry 0 rz 160 deg; joints [0.239, 59.542, -5.878, -155.407, 56.224, 165.724]
  Set speed (16.5 mm/s)
  Call Extruder(1214.90172)
  MoveL 7737 to (520.53, 453.73, 136) mm, rotated rx -180 ry 0 rz 160 deg; joints [0.327, 59.84, -6.472, -155.221, 55.978, 165.518]
  Set speed (16.5 mm/s)
  Call Extruder(1221.26526)
  MoveL 7738 to (522.21, 454.51, 136) mm, rotated rx -180 ry 0 rz 160 deg; joints [0.422, 60.132, -7.051, -155.028, 55.741, 165.31]
  Set speed (16.5 mm/s)
  Call Extruder(1227.44489)
  MoveL 7739 to (523.82, 455.34, 136) mm, rotated rx 180 ry 0 rz 160 deg; joints [0.52, 60.412, -7.608, -154.833, 55.516, 165.103]
  Set speed (16.5 mm/s)
  Call Extruder(1234.02326)
  MoveL 7740 to (525.5, 456.27, 136) mm, rotated rx 180 ry 0 rz 160 deg; joints [0.631, 60.708, -8.194, -154.617, 55.281, 164.878]
  Set speed (16.5 mm/s)
  Call Extruder(1240.29523)
  MoveL 7741 to (527.07, 457.22, 136) mm, rotated rx -180 ry 0 rz 160 deg; joints [0.743, 60.986, -8.747, -154.403, 55.063, 164.659]
  Set speed (16.5 mm/s)
  Call Extruder(1246.76503)
  MoveL 7742 to (528.65, 458.27, 136) mm, rotated rx 180 ry 0 rz 160 deg; joints [0.866, 61.27, -9.308, -154.174, 54.845, 164.428]
  Set speed (16.5 mm/s)
  Call Extruder(1253.04563)
  MoveL 7743 to (530.14, 459.33, 136) mm, rotated rx 180 ry 0 rz 160 deg; joints [0.991, 61.541, -9.845, -153.945, 54.64, 164.201]
  Set speed (16.5 mm/s)
  Call Extruder(1259.46602)
  MoveL 7744 to (531.63, 460.48, 136) mm, rotated rx 180 ry 0 rz 160 deg; joints [1.124, 61.813, -10.384, -153.703, 54.437, 163.965]
  Set speed (16.5 mm/s)
  Call Extruder(1265.83069)
  MoveL 7745 to (533.06, 461.67, 136) mm, rotated rx -180 ry 0 rz 160 deg; joints [1.262, 62.078, -10.909, -153.458, 54.243, 163.728]
  Set speed (16.5 mm/s)
  Call Extruder(1272.22080)
  MoveL 7746 to (534.45, 462.91, 136) mm, rotated rx -180 ry 0 rz 160 deg; joints [1.406, 62.339, -11.424, -153.205, 54.056, 163.487]
  Set speed (16.5 mm/s)
  Call Extruder(1278.40767)
  MoveL 7747 to (535.76, 464.17, 136) mm, rotated rx -180 ry 0 rz 160 deg; joints [1.55, 62.585, -11.912, -152.954, 53.883, 163.252]
  Set speed (16.5 mm/s)
  Call Extruder(1282.06716)
  MoveL 7748 to (536.51, 464.93, 136) mm, rotated rx -180 ry 0 rz 160 deg; joints [1.638, 62.728, -12.195, -152.804, 53.784, 163.112]
  Set speed (16.5 mm/s)
  Call Extruder(1285.52551)
  MoveL 7749 to (537.2, 465.67, 136) mm, rotated rx 180 ry 0 rz 160 deg; joints [1.722, 62.862, -12.458, -152.66, 53.693, 162.979]
  Set speed (16.5 mm/s)
  Call Extruder(1289.08786)
  MoveL 7750 to (537.9, 466.44, 136) mm, rotated rx 180 ry 0 rz 160 deg; joints [1.81, 62.997, -12.725, -152.51, 53.602, 162.841]
  Call Extruder(1292.67136)
  MoveL 7751 to (538.58, 467.23, 136) mm, rotated rx 180 ry 0 rz 160 deg; joints [1.901, 63.131, -12.989, -152.359, 53.513, 162.703]
  Call Extruder(1296.15163)
  MoveL 7752 to (539.24, 468.01, 136) mm, rotated rx -180 ry 0 rz 160 deg; joints [1.99, 63.258, -13.241, -152.21, 53.429, 162.568]
  Set speed (16.5 mm/s)
  Call Extruder(1300.49826)
  MoveL 7753 to (540.03, 469.01, 136) mm, rotated rx 180 ry 0 rz 160 deg; joints [2.103, 63.415, -13.55, -152.023, 53.329, 162.399]
  Set speed (16.5 mm/s)
  Call Extruder(1304.09656)
  MoveL 7754 to (540.66, 469.85, 136) mm, rotated rx -180 ry 0 rz 160 deg; joints [2.198, 63.542, -13.8, -151.866, 53.249, 162.259]
  Set speed (16.5 mm/s)
  Call Extruder(1306.89698)
  MoveL 7755 to (541.14, 470.51, 136) mm, rotated rx -180 ry 0 rz 160 deg; joints [2.273, 63.638, -13.991, -151.744, 53.189, 162.15]
  Set speed (16.5 mm/s)
  Call Extruder(1310.29871)
  MoveL 7756 to (541.72, 471.32, 136) mm, rotated rx 180 ry 0 rz 160 deg; joints [2.365, 63.754, -14.22, -151.594, 53.118, 162.017]
  Set speed (16.5 mm/s)
  Call Extruder(1313.21017)
  MoveL 7757 to (542.19, 472.03, 136) mm, rotated rx 180 ry 0 rz 160 deg; joints [2.445, 63.852, -14.411, -151.466, 53.06, 161.904]
  Set speed (16.5 mm/s)
  Call Extruder(1317.40707)
  MoveL 7758 to (542.86, 473.06, 136) mm, rotated rx -180 ry 0 rz 160 deg; joints [2.562, 63.989, -14.681, -151.279, 52.98, 161.741]
  Set speed (16.5 mm/s)
  Call Extruder(1321.00824)
  MoveL 7759 to (543.41, 473.96, 136) mm, rotated rx -180 ry 0 rz 160 deg; joints [2.663, 64.103, -14.907, -151.118, 52.914, 161.601]
  Set speed (16.5 mm/s)
  Call Extruder(1324.49156)
  MoveL 7760 to (543.93, 474.84, 136) mm, rotated rx -180 ry 0 rz 160 deg; joints [2.762, 64.211, -15.12, -150.962, 52.853, 161.466]
  Set speed (16.5 mm/s)
  Call Extruder(1328.05757)
  MoveL 7761 to (544.43, 475.75, 136) mm, rotated rx -180 ry 0 rz 160 deg; joints [2.864, 64.319, -15.332, -150.801, 52.795, 161.329]
  Set speed (16.5 mm/s)
  Call Extruder(1331.60626)
  MoveL 7762 to (544.92, 476.66, 136) mm, rotated rx -180 ry 0 rz 160 deg; joints [2.968, 64.423, -15.537, -150.641, 52.74, 161.193]
  Set speed (16.5 mm/s)
  Call Extruder(1335.10746)
  MoveL 7763 to (545.38, 477.57, 136) mm, rotated rx -180 ry 0 rz 160 deg; joints [3.07, 64.523, -15.735, -150.483, 52.688, 161.059]
  Set speed (16.5 mm/s)
  Call Extruder(1340.67942)
  MoveL 7764 to (546.08, 479.04, 136) mm, rotated rx -180 ry 0 rz 160 deg; joints [3.235, 64.677, -16.037, -150.23, 52.613, 160.847]
  Set speed (16.5 mm/s)
  Call Extruder(1346.56124)
  MoveL 7765 to (546.76, 480.62, 136) mm, rotated rx 180 ry 0 rz 160 deg; joints [3.412, 64.829, -16.336, -149.964, 52.544, 160.627]
  Set speed (16.5 mm/s)
  Call Extruder(1349.39227)
  MoveL 7766 to (547.07, 481.38, 136) mm, rotated rx 180 ry 0 rz 160 deg; joints [3.498, 64.9, -16.477, -149.835, 52.513, 160.521]
  Set speed (16.5 mm/s)
  Call Extruder(1356.36949)
  MoveL 7767 to (547.79, 483.3, 136) mm, rotated rx 180 ry 0 rz 160 deg; joints [3.713, 65.066, -16.802, -149.518, 52.447, 160.264]
  Set speed (16.5 mm/s)
  Call Extruder(1363.56778)
  MoveL 7768 to (548.44, 485.3, 136) mm, rotated rx 180 ry 0 rz 160 deg; joints [3.937, 65.224, -17.112, -149.192, 52.392, 160.004]
  Set speed (16.5 mm/s)
  Call Extruder(1370.65923)
  MoveL 7769 to (549, 487.29, 136) mm, rotated rx -180 ry 0 rz 160 deg; joints [4.161, 65.364, -17.389, -148.873, 52.352, 159.753]
  Set speed (16.5 mm/s)
  Call Extruder(1377.60933)
  MoveL 7770 to (549.47, 489.27, 136) mm, rotated rx -180 ry 0 rz 160 deg; joints [4.383, 65.489, -17.634, -148.562, 52.327, 159.514]
  Set speed (16.5 mm/s)
  Call Extruder(1384.79764)
  MoveL 7771 to (549.87, 491.33, 136) mm, rotated rx 180 ry 0 rz 160 deg; joints [4.615, 65.604, -17.859, -148.243, 52.314, 159.273]
  Call Extruder(1391.88991)
  MoveL 7772 to (550.19, 493.38, 136) mm, rotated rx -180 ry 0 rz 160 deg; joints [4.845, 65.702, -18.052, -147.932, 52.316, 159.043]
  Call Extruder(1399.05354)
  MoveL 7773 to (550.42, 495.46, 136) mm, rotated rx -180 ry 0 rz 160 deg; joints [5.08, 65.785, -18.216, -147.622, 52.332, 158.82]
  Call Extruder(1406.03966)
  MoveL 7774 to (550.56, 497.5, 136) mm, rotated rx -180 ry 0 rz 160 deg; joints [5.31, 65.852, -18.347, -147.324, 52.361, 158.611]
  Set speed (16.5 mm/s)
  Call Extruder(1413.11932)
  MoveL 7775 to (550.62, 499.57, 136) mm, rotated rx 180 ry 0 rz 160 deg; joints [5.545, 65.904, -18.45, -147.028, 52.405, 158.408]
  Set speed (16.5 mm/s)
  Call Extruder(1420.06534)
  MoveL 7776 to (550.6, 501.6, 136) mm, rotated rx -180 ry 0 rz 160 deg; joints [5.775, 65.94, -18.521, -146.743, 52.461, 158.219]
  Set speed (16.5 mm/s)
  Call Extruder(1427.27490)
  MoveL 7777 to (550.49, 503.71, 136) mm, rotated rx -180 ry 0 rz 160 deg; joints [6.015, 65.963, -18.564, -146.453, 52.533, 158.033]
  Call Extruder(1434.24927)
  MoveL 7778 to (550.29, 505.74, 136) mm, rotated rx -180 ry 0 rz 160 deg; joints [6.248, 65.968, -18.575, -146.18, 52.616, 157.865]
  Set speed (16.5 mm/s)
  Call Extruder(1441.55626)
  MoveL 7779 to (550.01, 507.86, 136) mm, rotated rx 180 ry 0 rz 160 deg; joints [6.492, 65.958, -18.555, -145.9, 52.716, 157.7]
  Set speed (16.5 mm/s)
  Call Extruder(1448.60728)
  MoveL 7780 to (549.65, 509.89, 136) mm, rotated rx 180 ry 0 rz 160 deg; joints [6.726, 65.932, -18.505, -145.638, 52.825, 157.552]
  Set speed (16.5 mm/s)
  Call Extruder(1455.98557)
  MoveL 7781 to (549.18, 511.99, 136) mm, rotated rx -180 ry 0 rz 160 deg; joints [6.971, 65.889, -18.419, -145.373, 52.954, 157.411]
  Set speed (16.5 mm/s)
  Call Extruder(1462.89666)
  MoveL 7782 to (548.66, 513.94, 136) mm, rotated rx -180 ry 0 rz 160 deg; joints [7.199, 65.833, -18.309, -145.132, 53.086, 157.291]
  Set speed (16.5 mm/s)
  Call Extruder(1469.82194)
  MoveL 7783 to (548.07, 515.88, 136) mm, rotated rx -180 ry 0 rz 160 deg; joints [7.427, 65.762, -18.17, -144.899, 53.23, 157.182]
  Set speed (16.5 mm/s)
  Call Extruder(1473.33827)
  MoveL 7784 to (547.73, 516.85, 136) mm, rotated rx -180 ry 0 rz 160 deg; joints [7.542, 65.72, -18.087, -144.784, 53.308, 157.132]
  Set speed (16.5 mm/s)
  Call Extruder(1476.89739)
  MoveL 7785 to (547.38, 517.83, 136) mm, rotated rx 180 ry 0 rz 160 deg; joints [7.658, 65.675, -17.999, -144.669, 53.388, 157.084]
  Set speed (16.5 mm/s)
  Call Extruder(1480.44231)
  MoveL 7786 to (547, 518.79, 136) mm, rotated rx 180 ry 0 rz 160 deg; joints [7.773, 65.625, -17.901, -144.558, 53.472, 157.04]
  Set speed (16.5 mm/s)
  Call Extruder(1483.94906)
  MoveL 7787 to (546.62, 519.74, 136) mm, rotated rx -180 ry 0 rz 160 deg; joints [7.887, 65.574, -17.8, -144.449, 53.557, 156.999]
  Set speed (16.5 mm/s)
  Call Extruder(1491.03714)
  MoveL 7788 to (545.77, 521.63, 136) mm, rotated rx -180 ry 0 rz 160 deg; joints [8.115, 65.457, -17.571, -144.237, 53.738, 156.925]
  Set speed (16.5 mm/s)
  Call Extruder(1495.29502)
  MoveL 7789 to (545.22, 522.75, 136) mm, rotated rx -180 ry 0 rz 160 deg; joints [8.251, 65.38, -17.419, -144.114, 53.852, 156.888]
  Set speed (16.5 mm/s)
  Call Extruder(1498.06845)
  MoveL 7790 to (544.85, 523.47, 136) mm, rotated rx -180 ry 0 rz 160 deg; joints [8.339, 65.327, -17.315, -144.036, 53.928, 156.866]
  Set speed (16.5 mm/s)
  Call Extruder(1501.59202)
  MoveL 7791 to (544.36, 524.38, 136) mm, rotated rx -180 ry 0 rz 160 deg; joints [8.45, 65.256, -17.177, -143.938, 54.026, 156.841]
  Set speed (16.5 mm/s)
  Call Extruder(1504.42416)
  MoveL 7792 to (543.96, 525.1, 136) mm, rotated rx 180 ry 0 rz 160 deg; joints [8.539, 65.197, -17.06, -143.862, 54.108, 156.824]
  Call Extruder(1508.76956)
  MoveL 7793 to (543.32, 526.2, 136) mm, rotated rx 180 ry 0 rz 160 deg; joints [8.675, 65.103, -16.875, -143.747, 54.234, 156.8]
  Set speed (16.5 mm/s)
  Call Extruder(1512.21436)
  MoveL 7794 to (542.79, 527.05, 136) mm, rotated rx -180 ry 0 rz 160 deg; joints [8.781, 65.024, -16.72, -143.658, 54.338, 156.785]
  Set speed (16.5 mm/s)
  Call Extruder(1515.77654)
  MoveL 7795 to (542.22, 527.93, 136) mm, rotated rx 180 ry 0 rz 160 deg; joints [8.891, 64.94, -16.554, -143.57, 54.447, 156.773]
  Set speed (16.5 mm/s)
  Call Extruder(1519.34583)
  MoveL 7796 to (541.63, 528.79, 136) mm, rotated rx -180 ry 0 rz 160 deg; joints [8.999, 64.851, -16.38, -143.483, 54.559, 156.764]
  Set speed (16.5 mm/s)
  Call Extruder(1522.80754)
  MoveL 7797 to (541.05, 529.62, 136) mm, rotated rx 180 ry 0 rz 160 deg; joints [9.104, 64.763, -16.206, -143.401, 54.669, 156.758]
  Call Extruder(1526.52765)
  MoveL 7798 to (540.41, 530.49, 136) mm, rotated rx 180 ry 0 rz 160 deg; joints [9.216, 64.664, -16.012, -143.316, 54.789, 156.755]
  Set speed (16.5 mm/s)
  Call Extruder(1529.87648)
  MoveL 7799 to (539.81, 531.27, 136) mm, rotated rx 180 ry 0 rz 160 deg; joints [9.316, 64.573, -15.833, -143.241, 54.899, 156.755]
  Set speed (16.5 mm/s)
  Call Extruder(1533.47537)
  MoveL 7800 to (539.15, 532.09, 136) mm, rotated rx -180 ry 0 rz 160 deg; joints [9.422, 64.472, -15.633, -143.163, 55.02, 156.759]
  Set speed (16.5 mm/s)
  Call Extruder(1536.99948)
  MoveL 7801 to (538.49, 532.88, 136) mm, rotated rx -180 ry 0 rz 160 deg; joints [9.525, 64.369, -15.431, -143.089, 55.14, 156.765]
  Set speed (16.5 mm/s)
  Call Extruder(1540.55785)
  MoveL 7802 to (537.8, 533.67, 136) mm, rotated rx 180 ry 0 rz 160 deg; joints [9.627, 64.263, -15.221, -143.018, 55.263, 156.775]
  Set speed (16.5 mm/s)
  Call Extruder(1544.23012)
  MoveL 7803 to (537.08, 534.46, 136) mm, rotated rx 180 ry 0 rz 160 deg; joints [9.732, 64.15, -14.999, -142.946, 55.392, 156.789]
  Set speed (16.5 mm/s)
  Call Extruder(1547.72780)
  MoveL 7804 to (536.38, 535.2, 136) mm, rotated rx 180 ry 0 rz 160 deg; joints [9.831, 64.04, -14.783, -142.88, 55.515, 156.804]
  Set speed (16.5 mm/s)
  Call Extruder(1551.16163)
  MoveL 7805 to (535.67, 535.92, 136) mm, rotated rx 180 ry 0 rz 160 deg; joints [9.927, 63.93, -14.565, -142.817, 55.639, 156.822]
  Call Extruder(1554.73358)
  MoveL 7806 to (534.92, 536.64, 136) mm, rotated rx 180 ry 0 rz 160 deg; joints [10.026, 63.812, -14.333, -142.755, 55.769, 156.844]
  Call Extruder(1558.21996)
  MoveL 7807 to (534.18, 537.34, 136) mm, rotated rx 180 ry 0 rz 160 deg; joints [10.121, 63.695, -14.102, -142.696, 55.897, 156.868]
  Set speed (16.5 mm/s)
  Call Extruder(1564.21291)
  MoveL 7808 to (532.87, 538.5, 136) mm, rotated rx 180 ry 0 rz 160 deg; joints [10.281, 63.487, -13.692, -142.6, 56.12, 156.916]
  Call Extruder(1568.98334)
  MoveL 7809 to (531.79, 539.39, 136) mm, rotated rx -180 ry 0 rz 160 deg; joints [10.407, 63.317, -13.357, -142.529, 56.301, 156.96]
  Call Extruder(0.00000)
  Set speed (16.5 mm/s)
  Call Extruder(3.54082)
  MoveL 7810 to (530.98, 540.03, 136) mm, rotated rx -180 ry 0 rz 160 deg; joints [10.497, 63.187, -13.101, -142.479, 56.436, 156.997]
  Set speed (16.5 mm/s)
  Call Extruder(7.74958)
  MoveL 7811 to (530, 540.78, 136) mm, rotated rx 180 ry 0 rz 160 deg; joints [10.604, 63.032, -12.794, -142.423, 56.598, 157.042]
  Set speed (16.5 mm/s)
  Call Extruder(11.27254)
  MoveL 7812 to (529.16, 541.38, 136) mm, rotated rx 180 ry 0 rz 160 deg; joints [10.692, 62.898, -12.531, -142.378, 56.735, 157.084]
  Set speed (16.5 mm/s)
  Call Extruder(14.03824)
  MoveL 7813 to (528.5, 541.84, 136) mm, rotated rx 180 ry 0 rz 160 deg; joints [10.76, 62.792, -12.321, -142.345, 56.844, 157.119]
  Call Extruder(17.63741)
  MoveL 7814 to (527.62, 542.42, 136) mm, rotated rx 180 ry 0 rz 160 deg; joints [10.847, 62.653, -12.046, -142.303, 56.985, 157.166]
  Set speed (16.5 mm/s)
  Call Extruder(22.09362)
  MoveL 7815 to (526.52, 543.12, 136) mm, rotated rx 180 ry 0 rz 160 deg; joints [10.952, 62.477, -11.698, -142.255, 57.162, 157.228]
  Call Extruder(28.20905)
  MoveL 7816 to (524.98, 544.03, 136) mm, rotated rx 180 ry 0 rz 160 deg; joints [11.093, 62.231, -11.211, -142.196, 57.406, 157.32]
  Set speed (16.5 mm/s)
  Call Extruder(31.78369)
  MoveL 7817 to (524.07, 544.53, 136) mm, rotated rx -180 ry 0 rz 160 deg; joints [11.173, 62.084, -10.922, -142.165, 57.55, 157.377]
  Set speed (16.5 mm/s)
  Call Extruder(37.55366)
  MoveL 7818 to (522.57, 545.31, 136) mm, rotated rx 180 ry 0 rz 160 deg; joints [11.298, 61.845, -10.448, -142.118, 57.783, 157.474]
  Set speed (16.5 mm/s)
  Call Extruder(42.28541)
  MoveL 7819 to (521.32, 545.91, 136) mm, rotated rx -180 ry 0 rz 160 deg; joints [11.397, 61.644, -10.05, -142.086, 57.977, 157.559]
  Set speed (16.5 mm/s)
  Call Extruder(45.30013)
  MoveL 7820 to (520.52, 546.27, 136) mm, rotated rx 180 ry 0 rz 160 deg; joints [11.459, 61.515, -9.795, -142.068, 58.1, 157.615]
  Set speed (16.5 mm/s)
  Call Extruder(49.44711)
  MoveL 7821 to (519.41, 546.75, 136) mm, rotated rx 180 ry 0 rz 160 deg; joints [11.542, 61.337, -9.442, -142.044, 58.269, 157.694]
  Set speed (16.5 mm/s)
  Call Extruder(56.50129)
  MoveL 7822 to (517.49, 547.51, 136) mm, rotated rx 180 ry 0 rz 160 deg; joints [11.676, 61.029, -8.832, -142.012, 58.558, 157.836]
  Set speed (16.5 mm/s)
  Call Extruder(63.86828)
  MoveL 7823 to (515.45, 548.21, 136) mm, rotated rx 180 ry 0 rz 160 deg; joints [11.809, 60.702, -8.183, -141.989, 58.861, 157.993]
  Set speed (16.5 mm/s)
  Call Extruder(70.63835)
  MoveL 7824 to (513.55, 548.77, 136) mm, rotated rx -180 ry 0 rz 160 deg; joints [11.923, 60.398, -7.579, -141.976, 59.14, 158.144]
  Set speed (16.5 mm/s)
  Call Extruder(74.36383)
  MoveL 7825 to (512.5, 549.05, 136) mm, rotated rx -180 ry 0 rz 160 deg; joints [11.982, 60.229, -7.244, -141.973, 59.293, 158.231]
  Set speed (16.5 mm/s)
  Call Extruder(77.86411)
  MoveL 7826 to (511.51, 549.3, 136) mm, rotated rx -180 ry 0 rz 160 deg; joints [12.037, 60.07, -6.928, -141.972, 59.437, 158.313]
  Set speed (16.5 mm/s)
  Call Extruder(85.17083)
  MoveL 7827 to (509.42, 549.74, 136) mm, rotated rx -180 ry 0 rz 160 deg; joints [12.143, 59.734, -6.261, -141.977, 59.737, 158.492]
  Set speed (16.5 mm/s)
  Call Extruder(92.12802)
  MoveL 7828 to (507.41, 550.08, 136) mm, rotated rx 180 ry 0 rz 160 deg; joints [12.235, 59.412, -5.621, -141.992, 60.021, 158.669]
  Set speed (16.5 mm/s)
  Call Extruder(99.00376)
  MoveL 7829 to (505.42, 550.33, 136) mm, rotated rx 180 ry 0 rz 160 deg; joints [12.318, 59.092, -4.984, -142.015, 60.301, 158.85]
  Set speed (16.5 mm/s)
  Call Extruder(106.26105)
  MoveL 7830 to (503.31, 550.51, 136) mm, rotated rx 180 ry 0 rz 160 deg; joints [12.396, 58.753, -4.308, -142.049, 60.594, 159.046]
  Call Extruder(113.39900)
  MoveL 7831 to (501.23, 550.61, 136) mm, rotated rx -180 ry 0 rz 160 deg; joints [12.462, 58.418, -3.641, -142.091, 60.88, 159.246]
  Call Extruder(120.37920)
  MoveL 7832 to (499.19, 550.62, 136) mm, rotated rx 180 ry 0 rz 160 deg; joints [12.518, 58.091, -2.988, -142.142, 61.157, 159.445]
  Set speed (10.0 mm/s)
  MoveL 7833 to (499.19, 550.62, 140) mm, rotated rx -180 ry 0 rz 160 deg; joints [12.518, 57.502, -2.808, -142.003, 60.834, 159.157]
  Set speed (120.0 mm/s)
  MoveL 7834 to (499.24, 548.91, 140) mm, rotated rx -180 ry 0 rz 160 deg; joints [12.309, 57.45, -2.705, -142.245, 60.8, 159.303]
  Set speed (16.6 mm/s)
  Call Extruder(127.06149)
  MoveL 7835 to (497.27, 548.84, 140) mm, rotated rx 180 ry 0 rz 160 deg; joints [12.352, 57.133, -2.076, -142.304, 61.062, 159.499]
  Set speed (16.6 mm/s)
  Call Extruder(134.15660)
  MoveL 7836 to (495.19, 548.68, 140) mm, rotated rx 180 ry 0 rz 160 deg; joints [12.389, 56.796, -1.408, -142.377, 61.337, 159.711]
  Set speed (16.6 mm/s)
  Call Extruder(140.89104)
  MoveL 7837 to (493.22, 548.44, 140) mm, rotated rx -180 ry 0 rz 160 deg; joints [12.414, 56.478, -0.776, -142.454, 61.595, 159.916]
  Set speed (16.6 mm/s)
  Call Extruder(147.56079)
  MoveL 7838 to (491.28, 548.13, 140) mm, rotated rx -180 ry 0 rz 160 deg; joints [12.428, 56.164, -0.152, -142.541, 61.845, 160.123]
  Set speed (16.6 mm/s)
  Call Extruder(154.56895)
  MoveL 7839 to (489.26, 547.72, 140) mm, rotated rx 180 ry 0 rz 160 deg; joints [12.432, 55.837, 0.499, -142.641, 62.104, 160.344]
  Set speed (16.6 mm/s)
  Call Extruder(161.32946)
  MoveL 7840 to (487.33, 547.25, 140) mm, rotated rx -180 ry 0 rz 160 deg; joints [12.426, 55.523, 1.123, -142.746, 62.349, 160.56]
  Set speed (16.6 mm/s)
  Call Extruder(167.90857)
  MoveL 7841 to (485.47, 546.71, 140) mm, rotated rx 180 ry 0 rz 160 deg; joints [12.41, 55.221, 1.726, -142.858, 62.583, 160.772]
  Set speed (16.6 mm/s)
  Call Extruder(174.79601)
  MoveL 7842 to (483.55, 546.07, 140) mm, rotated rx -180 ry 0 rz 160 deg; joints [12.382, 54.908, 2.35, -142.984, 62.822, 160.997]
  Set speed (16.6 mm/s)
  Call Extruder(181.53998)
  MoveL 7843 to (481.7, 545.36, 140) mm, rotated rx 180 ry 0 rz 160 deg; joints [12.344, 54.605, 2.954, -143.117, 63.051, 161.219]
  Set speed (16.6 mm/s)
  Call Extruder(185.11571)
  MoveL 7844 to (480.73, 544.95, 140) mm, rotated rx 180 ry 0 rz 160 deg; joints [12.319, 54.446, 3.271, -143.192, 63.169, 161.337]
  Set speed (16.6 mm/s)
  Call Extruder(188.35577)
  MoveL 7845 to (479.85, 544.57, 140) mm, rotated rx -180 ry 0 rz 160 deg; joints [12.295, 54.303, 3.556, -143.261, 63.275, 161.444]
  Set speed (16.6 mm/s)
  Call Extruder(191.74169)
  MoveL 7846 to (478.95, 544.15, 140) mm, rotated rx -180 ry 0 rz 160 deg; joints [12.267, 54.155, 3.852, -143.335, 63.385, 161.556]
  Set speed (16.6 mm/s)
  Call Extruder(196.72561)
  MoveL 7847 to (477.63, 543.5, 140) mm, rotated rx -180 ry 0 rz 160 deg; joints [12.22, 53.939, 4.283, -143.448, 63.543, 161.722]
  Set speed (16.6 mm/s)
  Call Extruder(202.11252)
  MoveL 7848 to (476.24, 542.75, 140) mm, rotated rx -180 ry 0 rz 160 deg; joints [12.163, 53.709, 4.743, -143.577, 63.71, 161.901]
  Set speed (16.6 mm/s)
  Call Extruder(205.36826)
  MoveL 7849 to (475.41, 542.28, 140) mm, rotated rx -180 ry 0 rz 160 deg; joints [12.125, 53.572, 5.017, -143.658, 63.809, 162.01]
  Set speed (16.6 mm/s)
  Call Extruder(208.84052)
  MoveL 7850 to (474.53, 541.76, 140) mm, rotated rx -180 ry 0 rz 160 deg; joints [12.082, 53.427, 5.308, -143.745, 63.913, 162.126]
  Set speed (16.6 mm/s)
  Call Extruder(212.17768)
  MoveL 7851 to (473.69, 541.24, 140) mm, rotated rx 180 ry 0 rz 160 deg; joints [12.037, 53.289, 5.584, -143.832, 64.01, 162.238]
  Set speed (16.6 mm/s)
  Call Extruder(215.65837)
  MoveL 7852 to (472.84, 540.68, 140) mm, rotated rx 180 ry 0 rz 160 deg; joints [11.988, 53.147, 5.869, -143.925, 64.111, 162.354]
  Set speed (16.6 mm/s)
  Call Extruder(219.11807)
  MoveL 7853 to (471.99, 540.1, 140) mm, rotated rx -180 ry 0 rz 160 deg; joints [11.937, 53.007, 6.149, -144.019, 64.209, 162.469]
  Call Extruder(222.59909)
  MoveL 7854 to (471.16, 539.51, 140) mm, rotated rx 180 ry 0 rz 160 deg; joints [11.882, 52.868, 6.428, -144.117, 64.305, 162.585]
  Set speed (16.6 mm/s)
  Call Extruder(225.81353)
  MoveL 7855 to (470.4, 538.94, 140) mm, rotated rx -180 ry 0 rz 160 deg; joints [11.829, 52.741, 6.682, -144.209, 64.392, 162.692]
  Set speed (16.6 mm/s)
  Call Extruder(229.19706)
  MoveL 7856 to (469.62, 538.33, 140) mm, rotated rx 180 ry 0 rz 160 deg; joints [11.771, 52.61, 6.945, -144.308, 64.482, 162.805]
  Set speed (16.6 mm/s)
  Call Extruder(232.61103)
  MoveL 7857 to (468.84, 537.7, 140) mm, rotated rx -180 ry 0 rz 160 deg; joints [11.709, 52.478, 7.208, -144.41, 64.571, 162.918]
  Call Extruder(235.97777)
  MoveL 7858 to (468.08, 537.06, 140) mm, rotated rx 180 ry 0 rz 160 deg; joints [11.645, 52.351, 7.464, -144.512, 64.657, 163.029]
  Set speed (16.6 mm/s)
  Call Extruder(239.43340)
  MoveL 7859 to (467.31, 536.39, 140) mm, rotated rx -180 ry 0 rz 160 deg; joints [11.578, 52.222, 7.723, -144.619, 64.743, 163.143]
  Set speed (16.6 mm/s)
  Call Extruder(242.74964)
  MoveL 7860 to (466.59, 535.73, 140) mm, rotated rx 180 ry 0 rz 160 deg; joints [11.51, 52.101, 7.967, -144.725, 64.824, 163.252]
  Set speed (16.6 mm/s)
  Call Extruder(245.83859)
  MoveL 7861 to (465.94, 535.1, 140) mm, rotated rx -180 ry 0 rz 160 deg; joints [11.445, 51.989, 8.191, -144.824, 64.897, 163.353]
  Set speed (16.6 mm/s)
  Call Extruder(249.62172)
  MoveL 7862 to (465.15, 534.32, 140) mm, rotated rx 180 ry 0 rz 160 deg; joints [11.362, 51.854, 8.461, -144.948, 64.984, 163.476]
  Set speed (16.6 mm/s)
  Call Extruder(252.96848)
  MoveL 7863 to (464.46, 533.61, 140) mm, rotated rx 180 ry 0 rz 160 deg; joints [11.286, 51.738, 8.696, -145.06, 65.059, 163.585]
  Set speed (16.6 mm/s)
  Call Extruder(256.05062)
  MoveL 7864 to (463.84, 532.94, 140) mm, rotated rx -180 ry 0 rz 160 deg; joints [11.213, 51.632, 8.909, -145.165, 65.127, 163.684]
  Set speed (16.6 mm/s)
  Call Extruder(259.82736)
  MoveL 7865 to (463.11, 532.11, 140) mm, rotated rx -180 ry 0 rz 160 deg; joints [11.122, 51.504, 9.165, -145.296, 65.207, 163.806]
  Call Extruder(263.18841)
  MoveL 7866 to (462.46, 531.36, 140) mm, rotated rx -180 ry 0 rz 160 deg; joints [11.038, 51.394, 9.387, -145.414, 65.275, 163.913]
  Set speed (16.6 mm/s)
  Call Extruder(266.62056)
  MoveL 7867 to (461.83, 530.58, 140) mm, rotated rx -180 ry 0 rz 160 deg; joints [10.95, 51.283, 9.611, -145.537, 65.344, 164.022]
  Call Extruder(270.01705)
  MoveL 7868 to (461.21, 529.79, 140) mm, rotated rx 180 ry 0 rz 160 deg; joints [10.86, 51.175, 9.827, -145.66, 65.409, 164.13]
  Set speed (16.6 mm/s)
  Call Extruder(273.41502)
  MoveL 7869 to (460.61, 528.99, 140) mm, rotated rx 180 ry 0 rz 160 deg; joints [10.768, 51.07, 10.039, -145.785, 65.472, 164.236]
  Set speed (16.6 mm/s)
  Call Extruder(275.86123)
  MoveL 7870 to (460.18, 528.41, 140) mm, rotated rx 180 ry 0 rz 160 deg; joints [10.7, 50.995, 10.189, -145.876, 65.516, 164.313]
  Set speed (16.6 mm/s)
  Call Extruder(280.23223)
  MoveL 7871 to (459.45, 527.36, 140) mm, rotated rx -180 ry 0 rz 160 deg; joints [10.576, 50.866, 10.45, -146.041, 65.591, 164.448]
  Call Extruder(282.64369)
  MoveL 7872 to (459.06, 526.76, 140) mm, rotated rx 180 ry 0 rz 160 deg; joints [10.505, 50.796, 10.591, -146.133, 65.631, 164.522]
  Set speed (16.6 mm/s)
  Call Extruder(286.97856)
  MoveL 7873 to (458.38, 525.69, 140) mm, rotated rx -180 ry 0 rz 160 deg; joints [10.376, 50.674, 10.837, -146.301, 65.7, 164.654]
  Set speed (16.6 mm/s)
  Call Extruder(293.71022)
  MoveL 7874 to (457.37, 523.98, 140) mm, rotated rx 180 ry 0 rz 160 deg; joints [10.169, 50.492, 11.205, -146.567, 65.8, 164.856]
  Set speed (16.6 mm/s)
  Call Extruder(297.32011)
  MoveL 7875 to (456.86, 523.05, 140) mm, rotated rx 180 ry 0 rz 160 deg; joints [10.054, 50.398, 11.393, -146.712, 65.849, 164.963]
  Set speed (16.6 mm/s)
  Call Extruder(300.61856)
  MoveL 7876 to (456.41, 522.19, 140) mm, rotated rx 180 ry 0 rz 160 deg; joints [9.947, 50.316, 11.559, -146.846, 65.892, 165.06]
  Set speed (16.6 mm/s)
  Call Extruder(304.61266)
  MoveL 7877 to (455.89, 521.14, 140) mm, rotated rx 180 ry 0 rz 160 deg; joints [9.815, 50.219, 11.755, -147.009, 65.941, 165.176]
  Set speed (16.6 mm/s)
  Call Extruder(310.81022)
  MoveL 7878 to (455.13, 519.48, 140) mm, rotated rx -180 ry 0 rz 160 deg; joints [9.605, 50.076, 12.043, -147.267, 66.01, 165.353]
  Call Extruder(317.72453)
  MoveL 7879 to (454.36, 517.6, 140) mm, rotated rx 180 ry 0 rz 160 deg; joints [9.363, 49.928, 12.343, -147.56, 66.076, 165.547]
  Call Extruder(324.33767)
  MoveL 7880 to (453.7, 515.77, 140) mm, rotated rx -180 ry 0 rz 160 deg; joints [9.125, 49.796, 12.609, -147.844, 66.131, 165.727]
  Set speed (16.6 mm/s)
  Call Extruder(327.92542)
  MoveL 7881 to (453.37, 514.76, 140) mm, rotated rx -180 ry 0 rz 160 deg; joints [8.993, 49.73, 12.743, -147.999, 66.156, 165.823]
  Set speed (16.6 mm/s)
  Call Extruder(331.31726)
  MoveL 7882 to (453.08, 513.81, 140) mm, rotated rx -180 ry 0 rz 160 deg; joints [8.867, 49.669, 12.865, -148.147, 66.178, 165.913]
  Set speed (16.6 mm/s)
  Call Extruder(337.95947)
  MoveL 7883 to (452.57, 511.92, 140) mm, rotated rx -180 ry 0 rz 160 deg; joints [8.615, 49.56, 13.086, -148.44, 66.211, 166.085]
  Set speed (16.6 mm/s)
  Call Extruder(340.45916)
  MoveL 7884 to (452.39, 511.21, 140) mm, rotated rx 180 ry 0 rz 160 deg; joints [8.519, 49.522, 13.164, -148.551, 66.222, 166.148]
  Set speed (16.6 mm/s)
  Call Extruder(345.52975)
  MoveL 7885 to (452.07, 509.76, 140) mm, rotated rx 180 ry 0 rz 160 deg; joints [8.323, 49.449, 13.311, -148.776, 66.239, 166.274]
  Set speed (16.6 mm/s)
  Call Extruder(351.76579)
  MoveL 7886 to (451.74, 507.95, 140) mm, rotated rx 180 ry 0 rz 160 deg; joints [8.077, 49.369, 13.474, -149.056, 66.251, 166.426]
  Set speed (16.6 mm/s)
  Call Extruder(358.55645)
  MoveL 7887 to (451.45, 505.97, 140) mm, rotated rx -180 ry 0 rz 160 deg; joints [7.805, 49.293, 13.627, -149.362, 66.255, 166.586]
  Set speed (16.6 mm/s)
  Call Extruder(365.35691)
  MoveL 7888 to (451.25, 503.98, 140) mm, rotated rx -180 ry 0 rz 160 deg; joints [7.529, 49.229, 13.757, -149.67, 66.247, 166.74]
  Call Extruder(371.94770)
  MoveL 7889 to (451.13, 502.05, 140) mm, rotated rx 180 ry 0 rz 160 deg; joints [7.259, 49.179, 13.858, -149.969, 66.23, 166.884]
  Set speed (16.6 mm/s)
  Call Extruder(378.91067)
  MoveL 7890 to (451.08, 500, 140) mm, rotated rx 180 ry 0 rz 160 deg; joints [6.971, 49.138, 13.941, -150.285, 66.202, 167.03]
  Set speed (16.6 mm/s)
  Call Extruder(384.14151)
  MoveL 7891 to (451.11, 498.46, 140) mm, rotated rx 180 ry 0 rz 160 deg; joints [6.754, 49.116, 13.985, -150.521, 66.172, 167.136]
  Set speed (16.6 mm/s)
  Call Extruder(390.96130)
  MoveL 7892 to (451.21, 496.45, 140) mm, rotated rx -180 ry 0 rz 160 deg; joints [6.469, 49.099, 14.019, -150.829, 66.124, 167.268]
  Call Extruder(397.20684)
  MoveL 7893 to (451.38, 494.62, 140) mm, rotated rx -180 ry 0 rz 160 deg; joints [6.208, 49.094, 14.029, -151.109, 66.071, 167.384]
  Set speed (16.6 mm/s)
  Call Extruder(403.32586)
  MoveL 7894 to (451.62, 492.84, 140) mm, rotated rx 180 ry 0 rz 160 deg; joints [5.952, 49.1, 14.018, -151.381, 66.011, 167.492]
  Call Extruder(409.52955)
  MoveL 7895 to (451.92, 491.03, 140) mm, rotated rx 180 ry 0 rz 160 deg; joints [5.692, 49.116, 13.986, -151.654, 65.941, 167.596]
  Set speed (16.6 mm/s)
  Call Extruder(415.50363)
  MoveL 7896 to (452.27, 489.31, 140) mm, rotated rx 180 ry 0 rz 160 deg; joints [5.444, 49.141, 13.934, -151.915, 65.864, 167.691]
  Set speed (16.6 mm/s)
  Call Extruder(421.68143)
  MoveL 7897 to (452.7, 487.55, 140) mm, rotated rx 180 ry 0 rz 160 deg; joints [5.189, 49.177, 13.861, -152.18, 65.777, 167.784]
  Set speed (16.6 mm/s)
  Call Extruder(427.79772)
  MoveL 7898 to (453.19, 485.81, 140) mm, rotated rx -180 ry 0 rz 160 deg; joints [4.938, 49.223, 13.769, -152.44, 65.683, 167.871]
  Set speed (16.6 mm/s)
  Call Extruder(433.91071)
  MoveL 7899 to (453.74, 484.1, 140) mm, rotated rx -180 ry 0 rz 160 deg; joints [4.689, 49.278, 13.656, -152.695, 65.581, 167.952]
  Set speed (16.6 mm/s)
  Call Extruder(440.10560)
  MoveL 7900 to (454.37, 482.39, 140) mm, rotated rx -180 ry 0 rz 160 deg; joints [4.44, 49.345, 13.521, -152.948, 65.468, 168.029]
  Set speed (16.6 mm/s)
  Call Extruder(446.24633)
  MoveL 7901 to (455.05, 480.71, 140) mm, rotated rx 180 ry 0 rz 160 deg; joints [4.197, 49.421, 13.367, -153.193, 65.348, 168.099]
  Set speed (16.6 mm/s)
  Call Extruder(452.27263)
  MoveL 7902 to (455.78, 479.1, 140) mm, rotated rx 180 ry 0 rz 160 deg; joints [3.962, 49.505, 13.198, -153.429, 65.223, 168.162]
  Call Extruder(458.47014)
  MoveL 7903 to (456.59, 477.46, 140) mm, rotated rx 180 ry 0 rz 160 deg; joints [3.724, 49.601, 13.003, -153.665, 65.087, 168.222]
  Set speed (16.6 mm/s)
  Call Extruder(464.36656)
  MoveL 7904 to (457.42, 475.94, 140) mm, rotated rx 180 ry 0 rz 160 deg; joints [3.503, 49.702, 12.8, -153.883, 64.949, 168.273]
  Call Extruder(470.43826)
  MoveL 7905 to (458.33, 474.4, 140) mm, rotated rx 180 ry 0 rz 160 deg; joints [3.279, 49.815, 12.572, -154.101, 64.8, 168.32]
  Set speed (16.6 mm/s)
  Call Extruder(476.72555)
  MoveL 7906 to (459.32, 472.84, 140) mm, rotated rx -180 ry 0 rz 160 deg; joints [3.053, 49.941, 12.317, -154.32, 64.639, 168.362]
  Call Extruder(482.84807)
  MoveL 7907 to (460.35, 471.36, 140) mm, rotated rx -180 ry 0 rz 160 deg; joints [2.839, 50.073, 12.05, -154.524, 64.474, 168.398]
  Set speed (16.6 mm/s)
  Call Extruder(488.78907)
  MoveL 7908 to (461.4, 469.96, 140) mm, rotated rx -180 ry 0 rz 160 deg; joints [2.637, 50.209, 11.775, -154.715, 64.308, 168.426]
  Set speed (16.6 mm/s)
  Call Extruder(495.00470)
  MoveL 7909 to (462.55, 468.54, 140) mm, rotated rx -180 ry 0 rz 160 deg; joints [2.432, 50.361, 11.468, -154.906, 64.127, 168.45]
  Set speed (16.6 mm/s)
  Call Extruder(501.19084)
  MoveL 7910 to (463.75, 467.16, 140) mm, rotated rx -180 ry 0 rz 160 deg; joints [2.235, 50.521, 11.146, -155.088, 63.94, 168.468]
  Call Extruder(507.23747)
  MoveL 7911 to (464.97, 465.87, 140) mm, rotated rx -180 ry 0 rz 160 deg; joints [2.049, 50.685, 10.814, -155.256, 63.751, 168.479]
  Set speed (16.6 mm/s)
  Call Extruder(513.29231)
  MoveL 7912 to (466.24, 464.61, 140) mm, rotated rx -180 ry 0 rz 160 deg; joints [1.87, 50.858, 10.466, -155.415, 63.556, 168.484]
  Set speed (16.6 mm/s)
  Call Extruder(519.54374)
  MoveL 7913 to (467.59, 463.37, 140) mm, rotated rx 180 ry 0 rz 160 deg; joints [1.693, 51.044, 10.091, -155.57, 63.349, 168.483]
  Call Extruder(525.75103)
  MoveL 7914 to (468.98, 462.18, 140) mm, rotated rx -180 ry 0 rz 160 deg; joints [1.525, 51.237, 9.702, -155.714, 63.137, 168.476]
  Set speed (16.6 mm/s)
  Call Extruder(531.96824)
  MoveL 7915 to (470.42, 461.05, 140) mm, rotated rx 180 ry 0 rz 160 deg; joints [1.365, 51.438, 9.298, -155.847, 62.92, 168.462]
  Set speed (16.6 mm/s)
  Call Extruder(537.31924)
  MoveL 7916 to (471.68, 460.11, 140) mm, rotated rx -180 ry 0 rz 160 deg; joints [1.234, 51.617, 8.938, -155.953, 62.728, 168.445]
  Set speed (16.6 mm/s)
  Call Extruder(544.04960)
  MoveL 7917 to (473.32, 459, 140) mm, rotated rx 180 ry 0 rz 160 deg; joints [1.079, 51.85, 8.47, -156.075, 62.482, 168.416]
  Set speed (16.6 mm/s)
  Call Extruder(550.22905)
  MoveL 7918 to (474.87, 458.04, 140) mm, rotated rx 180 ry 0 rz 160 deg; joints [0.945, 52.071, 8.026, -156.176, 62.252, 168.383]
  Set speed (16.6 mm/s)
  Call Extruder(556.34738)
  MoveL 7919 to (476.43, 457.14, 140) mm, rotated rx -180 ry 0 rz 160 deg; joints [0.821, 52.296, 7.575, -156.266, 62.019, 168.344]
  Set speed (16.6 mm/s)
  Call Extruder(562.45432)
  MoveL 7920 to (478.02, 456.31, 140) mm, rotated rx 180 ry 0 rz 160 deg; joints [0.706, 52.527, 7.111, -156.344, 61.783, 168.298]
  Set speed (16.6 mm/s)
